// ---------------------------------------------------------------------------
// transition condition
      A     M    151.6; // Amount
      O     M    120.6;
      A     #S2I.SFM39.I01; // Released
      AN    M    102.2;
      =     M    102.1;

// subphase evaluation
      L     MW   110;
      JL    A300;
      JU    COMM; // subphase  0:
      JU    A301; // subphase  1: Gully VEE
      JU    A302; // subphase  2: Gully Befüllung
// ---------------------------------------------------------------------------
A300: SET   ;
      S     M    110.7; // Error unknown subphase
      JU    COMM;
// subphase 1: Gully VEE
A301: SET   ;
// -------------------------------------------------
// subphase timer & counter
      A     M    103.0;

// -------------------------------------------------
// subphase actuator
      A     M    103.3;

// -------------------------------------------------
// subphase transition
      SET   ;
      =     M    103.1;
      JU    COMM;
// subphase 2: Gully Befüllung
A302: SET   ;
// -------------------------------------------------
// subphase timer & counter
      A     M    103.0;

// -------------------------------------------------
// subphase actuator
      A     M    103.3;

// -------------------------------------------------
// subphase transition
      CLR   ;
      =     M    103.1;
      JU    COMM;

NETWORK
TITLE =phase 4: Fill System
//SFM   Use                                 Datatype        UoM
//----+-------------------------------------------------------------------------
// 00 : Watch Dog Time                      Duration        min
// 20 : Flow                                Value           l/h
// 41 : Amount                              Value           kg
X4:   SET   ;
// ---------------------------------------------------------------------------
// General CM evaluation
      CALL FC   120 (
           ChkType                  := 3,
           ChkOK                    := #ChkOK);

      AN    #ChkOK;
      S     M    120.3;

// ---------------------------------------------------------------------------
// general functions
      AN    M    121.2;
      A     M    102.3;
      =     #RRel;


// ---------------------------------------------------------------------------
// messages
// ---------------------------------------------------------------------------
// timer & counter
      A     M    102.0;

// ---------------------------------------------------------------------------
// pause timer
// ---------------------------------------------------------------------------
// communication

// ---------------------------------------------------------------------------
// control modules
      A     M    102.3;

// ---------------------------------------------------------------------------
// transition condition
      A     #SubStepMaxD;
      =     M    102.1;

// subphase evaluation
      L     MW   110;
      JL    A400;
      JU    COMM; // subphase  0:
// ---------------------------------------------------------------------------
A400: SET   ;
      S     M    110.7; // Error unknown subphase
      JU    COMM;

NETWORK
TITLE =phase 5: Transfer
//SFM   Use                                 Datatype        UoM
//----+-------------------------------------------------------------------------
// 00 : Watch Dog Time                      Duration        min
// 20 : Flow                                Value           l/h
// 41 : Amount                              Value           kg
X5:   SET   ;
// ---------------------------------------------------------------------------
// General CM evaluation
      CALL FC   120 (
           ChkType                  := 3,
           ChkOK                    := #ChkOK);

      AN    #ChkOK;
      S     M    120.3;

      CALL FC   779 (
           P1Sel                    := #U.Seq.SFM[11].Sp,
           P2Sel                    := #U.Seq.SFM[12].Sp,
           P3Sel                    := #U.Seq.SFM[13].Sp,
           P1Rel                    := DB125.DBX  363.2,
           P2Rel                    := DB125.DBX  411.2,
           P3Rel                    := DB125.DBX  459.2,
           CurrSel                  := #U.Seq.User.Real10);

// ---------------------------------------------------------------------------
// general functions
      AN    M    121.2;
      A     M    102.3;
      =     #RRel;

      A     M    102.3;
      =     DB125.DBX   26.3;

      A     M    102.3;
      =     DB125.DBX   27.2;

// ---------------------------------------------------------------------------
// messages

      AN    #ComDST;
      JCN   N501;
      L     903; // Destination not Ready
      T     MD    90;
N501: NOP   0;

// ---------------------------------------------------------------------------
// timer & counter

// Amount
      AN    #U.Seq.SFM[16].P;
      =     #xTmp;
      CALL FC   710 (
           RefVal                   := DB125.DBD  230,
           Active                   := #xTmp,
           Reset                    := #U.Seq.SFM[16].Res,
           Down                     := FALSE,
           CntVal                   := #U.Seq.SFM[16].Val,
           RefMem                   := #U.Seq.User.Real2);

      AN    #U.Seq.SFM[17].P; // TT Counter
      =     #xTmp;
      CALL FC   710 (
           RefVal                   := DB125.DBD  230,
           Active                   := #xTmp,
           Reset                    := #U.Seq.SFM[17].Res,
           Down                     := FALSE,
           CntVal                   := #U.Seq.SFM[17].Val,
           RefMem                   := #U.Seq.User.Real4);

// ---------------------------------------------------------------------------
// pause timer
// ---------------------------------------------------------------------------
// communication


// ---------------------------------------------------------------------------
// Check Partner
      AN    #ComSRC;
      O(    ;
      AN    DB125.DBX  218.3;
      AN    DB125.DBX  218.4;
      )     ;
      AN    #U.Seq.Step0;
      AN    #CIP;
      JCN   NC05;
      L     904; // "Source Not Ready!
      T     MD    90;
NC05: NOP   0;

      AN    DB125.DBX  314.0; // Water Tank Ready
      AN    DB125.DBX  314.1;
      AN    #ComDST;
      A     #S2I.SFM10.I00;
      AN    #U.Seq.Step0;
      AN    #U.Seq.PO.B22;
      AN    #CIP;
      JCN   NX05;
      L     903; // Destination not Ready
      T     MD    90;
NX05: NOP   0;

// ---------------------------------------------------------------------------
// control modules
      A     M    102.3;

// ---------------------------------------------------------------------------
// transition condition
      L     #U.Seq.User.Real10;
      L     0.000000e+000;
      ==R   ;
      O     M    151.7; // Amount
      AN    M    102.2;
      =     M    102.1;
// subphase repeat function
      A     #SubStepMax;
      JCN   Y5;
      L     1;
      T     MW   116;
Y5:   SET   ;
// ---------------------------------------------------------------------------
// ---------------------------------------------------------------------------
// subphase evaluation
      L     MW   110;
      JL    A500;
      JU    COMM; // subphase  0:
      JU    A501; // subphase  1: Waiting
      JU    A502; // subphase  2: Active
      JU    A503; // subphase  3: Tank Change
// ---------------------------------------------------------------------------
A500: SET   ;
      S     M    110.7; // Error unknown subphase
      JU    COMM;

// subphase 1: Waiting
A501: SET   ;

// -------------------------------------------------
// subphase timer & counter
      A     M    103.0;

// -------------------------------------------------
// subphase actuator
      A     M    103.3;

// -------------------------------------------------
// subphase transition
      A(    ;
      L     #U.Seq.User.Real10;
      L     #U.Seq.SFM[10].Sp;
      <>R   ;
      )     ;
      O(    ;
      A     DB125.DBX  314.0;
      A     DB125.DBX  315.2;
      A     DB125.DBX  218.3;
      O     #S2I.SFM10.I00;
      )     ;
      =     M    103.1;

      JU    COMM;

// subphase 2: Active
A502: SET   ;

// Well Management
      A     DB125.DBX  314.1;
      A     #ComSRC; // Comms Well Managment
      A     M    103.3;
      =     DB125.DBX   26.1; // Request Water

// Water Tank
      A     DB125.DBX  218.3; // Well Managment
      O     DB125.DBX  218.4; // Well Managment
      A     M    103.3;
      =     DB125.DBX   26.4;

// -------------------------------------------------
// subphase timer & counter
      A     M    103.0;
// -------------------------------------------------
// subphase actuator
      L     #U.Seq.SFM[22].Sp;
      L     1.000000e+001;
      <R    ;
      A(    ;
      L     #U.Seq.SFM[22].Sp;
      L     5.000000e+000;
      >R    ;
      )     ;
      A     DB125.DBX  314.1;
      A     DB125.DBX  219.7;
      A     M    103.3;
      =     DB220.DBX  348.0;
      =     DB220.DBX  188.0;
      =     DB220.DBX  268.0;
// -------------------------------------------------
// subphase transition
      L     #U.Seq.User.Real10;
      L     #U.Seq.SFM[10].Sp;
      <>R   ;
      O     #S2I.SFM10.I00;
      ON    DB125.DBX  315.2;
      =     M    103.1;

      JU    COMM;
// subphase 3: Tank Change
A503: SET   ;
      L     #U.Seq.User.Real10;
      T     #U.Seq.SFM[10].Sp; // Current Tank

// -------------------------------------------------
// subphase timer & counter
      A     M    103.0;
      =     M    162.0;

// -------------------------------------------------
// subphase actuator
//      A     "U099ComD".Own.Bit26
//      A     "SOSPH"
//      =     "C02ActD".A_G1.ACo
// -------------------------------------------------
// subphase transition
      AN    #S2I.SFM10.I00;
      AN    M    102.2;
      =     M    103.1;
      JU    COMM;
NETWORK
TITLE =phase 6: Standby
//SFM   Use                                 Datatype        UoM
//----+-------------------------------------------------------------------------
// 00 : Watch Dog Time                      Duration        min
// 02 : Step Time                           Duration        h
X6:   SET   ;
// ---------------------------------------------------------------------------
// General CM evaluation
      CALL FC   120 (
           ChkType                  := 3,
           ChkOK                    := #ChkOK);

      AN    #ChkOK;
      S     M    120.3;


      CALL FC   779 (
           P1Sel                    := #U.Seq.SFM[11].Sp,
           P2Sel                    := #U.Seq.SFM[12].Sp,
           P3Sel                    := #U.Seq.SFM[13].Sp,
           P1Rel                    := DB125.DBX  363.2,
           P2Rel                    := DB125.DBX  411.2,
           P3Rel                    := DB125.DBX  459.2,
           CurrSel                  := #U.Seq.User.Real10);

      L     #U.Seq.User.Real10;
      T     #U.Seq.SFM[10].Sp;

// ---------------------------------------------------------------------------
// general functions
      AN    M    121.2;
      A     M    102.3;
      =     #RRel;
      R     DB125.DBX   26.1;

      A     M    102.3;
      =     DB125.DBX   27.2;
// ---------------------------------------------------------------------------
// messages
      AN    M    151.7;
      A     M    150.1; // Max Standby Time
      JCN   N601;
      L     919; // "Press Start to Continue"
      T     MD    90;
N601: NOP   0;

// ---------------------------------------------------------------------------
// timer & counter
      A     M    102.0;
      =     M    130.1;
// ---------------------------------------------------------------------------
// pause timer
//      ON    "SOPH"
//      O     "SFM02D"
//      S     "SFM02P"                    // Step Time

      SET   ;
      S     M    141.7;

// ---------------------------------------------------------------------------
// communication

// ---------------------------------------------------------------------------
// Check Partner
      AN    #ComSRC;
      O(    ;
      AN    DB125.DBX  218.3;
      AN    DB125.DBX  218.4;
      )     ;
      AN    #U.Seq.Step0;
      AN    #CIP;
      JCN   NC06;
      L     904; // "Source Not Ready!
      T     MD    90;
NC06: NOP   0;

//      AN    "C02ComD".DST.WfFi          // Water Tank Ready
//      AN    "C02ComD".DST.Fill
      AN    #ComDST;
      AN    M    150.1; // Max Standby Time
//      A     #S2I.SFM10.I00
      AN    M    151.7;
      CLR   ; // Thats why we are in StandBy
      JCN   NX06;
      L     903; // Destination not Ready
      T     MD    90;
NX06: NOP   0;

// ---------------------------------------------------------------------------
// control modules

// ---------------------------------------------------------------------------
// transition condition
      CLR   ;
      =     #xTmp;

      AN    #S2I.SFM10.I00;
      AN    M    150.1; // Max Standby Time
      AN    M    151.7;
      S     #xTmp; // AutoCont
      JCN   N6x2;
      L     MW   104;
      L     -1;
      +I    ;
      T     MW   106;
N6x2: NOP   0;

      A     M    150.1; // Max Standby Time
      AN    M    151.7;
      A     M    120.6;
      S     #xTmp; // ReqRestart
      JCN   N6y2;
      L     MW   104;
      L     -2;
      +I    ;
      T     MW   106;
N6y2: NOP   0;

      A     M    150.1; // Max Standby Time
      A     M    151.7;
      S     #xTmp; // ReqEnd

      A     #xTmp;
      AN    M    102.2;
      =     M    102.1;

// subphase evaluation
      L     MW   110;
      JL    A600;
      JU    COMM; // subphase  0:
// ---------------------------------------------------------------------------
A600: SET   ;
      S     M    110.7; // Error unknown subphase
      JU    COMM;
NETWORK
TITLE =phase 8: Push Out
//SFM   Use                                 Datatype        UoM
//----+-------------------------------------------------------------------------
// 00 : Watch Dog Time                      Duration        min
// 20 : Flow                                Value           l/h
// 41 : Amount                              Value           kg
X8:   SET   ;
// ---------------------------------------------------------------------------
// General CM evaluation
      CALL FC   120 (
           ChkType                  := 3,
           ChkOK                    := #ChkOK);

      AN    #ChkOK;
      S     M    120.3;

// ---------------------------------------------------------------------------
// general functions
      AN    M    121.2;
      A     M    102.3;
      =     #RRel;

// ---------------------------------------------------------------------------
// messages
// ---------------------------------------------------------------------------
// timer & counter
      A     M    102.0;

// ---------------------------------------------------------------------------
// pause timer
// ---------------------------------------------------------------------------
// communication

// ---------------------------------------------------------------------------
// control modules
      A     M    102.3;

// ---------------------------------------------------------------------------
// transition condition
      A     #SubStepMaxD;
      =     M    102.1;

// subphase evaluation
      L     MW   110;
      JL    A800;
      JU    COMM; // subphase  0:
// ---------------------------------------------------------------------------
A800: SET   ;
      S     M    110.7; // Error unknown subphase
      JU    COMM;
NETWORK
TITLE =phase 11: Postrinse
//SFM   Use                                 Datatype        UoM
//----+-------------------------------------------------------------------------
// 00 : Watch Dog Time                      Duration        min
// 20 : Flow                                Value           l/h
// 41 : Amount                              Value           kg
X11:  SET   ;
// ---------------------------------------------------------------------------
// General CM evaluation
      CALL FC   120 (
           ChkType                  := 3,
           ChkOK                    := #ChkOK);

      AN    #ChkOK;
      S     M    120.3;

// ---------------------------------------------------------------------------
// general functions
      AN    M    121.2;
      A     M    102.3;
      =     #RRel;

// ---------------------------------------------------------------------------
// messages
// ---------------------------------------------------------------------------
// timer & counter
      A     M    102.0;

// ---------------------------------------------------------------------------
// pause timer
// ---------------------------------------------------------------------------
// communication

// ---------------------------------------------------------------------------
// control modules
      A     M    102.3;

// ---------------------------------------------------------------------------
// transition condition
      A     #SubStepMaxD;
      =     M    102.1;

// subphase evaluation
      L     MW   110;
      JL    B100;
      JU    COMM; // subphase  0:
// ---------------------------------------------------------------------------
B100: SET   ;
      S     M    110.7; // Error unknown subphase
      JU    COMM;
NETWORK
TITLE =phase 21: Prepare Line
//SFM   Use                                 Datatype        UoM
//----+-------------------------------------------------------------------------
// 00 : Watch Dog Time                      Duration        min
X21:  SET   ;
// ---------------------------------------------------------------------------
// General CM evaluation
      CALL FC   120 (
           ChkType                  := 3,
           ChkOK                    := #ChkOK);

      AN    #ChkOK;
      S     M    120.3;

      A     M    102.2;
      JCN   N903;
      L     DB125.DBD  234;
      T     #U.Seq.SFM[22].Sp;
N903: NOP   0;
// ---------------------------------------------------------------------------
// general functions
      AN    M    121.2;
      A     M    102.3;
      =     #RRel;

// ---------------------------------------------------------------------------
// messages
// ---------------------------------------------------------------------------
// timer & counter
      A     M    102.0;

// ---------------------------------------------------------------------------
// pause timer
// ---------------------------------------------------------------------------
// communication
      A     #ComSRC;
      A     M    103.3;
      =     DB125.DBX   26.0; // Wait for filling
      =     DB125.DBX   27.2;
// ---------------------------------------------------------------------------
// control modules
      A     M    102.3;

// ---------------------------------------------------------------------------
// transition condition
      A     #SubStepMaxD;
      AN    M    102.2;
      =     M    102.1;

// ---------------------------------------------------------------------------
// ---------------------------------------------------------------------------
// subphase repeat function
//      A     #SubStepMax
//      JCN  Y21
//      L     1
//      T     "SOSubStepNew"
//Y21:  SET

// subphase evaluation
      L     MW   110;
      JL    C100;
      JU    COMM; // subphase  0:
      JU    C101; // subphase  1: Start Well
      JU    C102; // subphase  2: Check Partner
// ---------------------------------------------------------------------------
C100: SET   ;
      S     M    110.7; // Error unknown subphase
      JU    COMM;

// subphase 1: Start Well
C101: SET   ;
// Request Well start

// -------------------------------------------------
// subphase timer & counter
      A     M    103.0;

// -------------------------------------------------
// subphase actuator
      A     M    103.3;

// -------------------------------------------------
// subphase transition
      A     DB125.DBX  218.3; // Well Ready
      A     #ComSRC;
      AN    M    103.2;
      =     M    103.1;
      JU    COMM;

// subphase 2: Check Partner
C102: SET   ;
      A     M    103.3;
      =     DB125.DBX   26.3;
// -------------------------------------------------
// subphase timer & counter
      A     M    103.0;

// -------------------------------------------------
// subphase actuator
      AN    DB125.DBX   75.2; // Swingbend drain Tank filling
      JCN   N801;
      L     920; // Check connections (Swingbend)
      T     MD    90;
N801: NOP   0;

// -------------------------------------------------
// subphase transition
      A     DB125.DBX   75.2; // Swingbend drain Tank filling
      A     DB125.DBX  218.3; // Well Ready
      A     #ComSRC; // Communication Well Management
      AN    M    103.2;
      =     M    103.1;
      JU    COMM;
NETWORK
TITLE =phase 22: Tank Selection
//SFM   Use                                 Datatype        UoM
//----+-------------------------------------------------------------------------
// 00 : Watch Dog Time                      Duration        min
X22:  SET   ;
// ---------------------------------------------------------------------------
// General CM evaluation
      CALL FC   120 (
           ChkType                  := 3,
           ChkOK                    := #ChkOK);

      AN    #ChkOK;
      S     M    120.3;

// ---------------------------------------------------------------------------
// general functions
      AN    M    121.2;
      A     M    102.3;
      =     #RRel;

// ---------------------------------------------------------------------------
// messages

      AN    #S2I.SFM11.I00; // Priority 1 Tank
      A     #ComSRC;
      JCN   N901;
      L     919; // "Press Start to Continue"
      T     MD    90;
N901: NOP   0;

// ---------------------------------------------------------------------------
// timer & counter
      A     M    102.0;

// ---------------------------------------------------------------------------
// pause timer
// ---------------------------------------------------------------------------
// communication
      A     M    102.0;
      R     DB125.DBX   26.1;
      A     M    102.0;
      =     DB125.DBX   26.0;

// ---------------------------------------------------------------------------
// control modules
      A     M    102.3;

// ---------------------------------------------------------------------------
// transition condition
      A     M    120.6;
      A     #ComSRC;
      AN    M    102.2;
      =     M    102.1;

// subphase evaluation
      L     MW   110;
      JL    C200;
      JU    COMM; // subphase  0:
// ---------------------------------------------------------------------------
C200: SET   ;
      S     M    110.7; // Error unknown subphase
      JU    COMM;

NETWORK
TITLE =End Of Sequence Organisation

COMM: SET   ;

// ---------------------------------------------------------------------------
// Comm with Transfer Plan Unit
      AN    DB125.DBX  509.0;
      R     DB125.DBX   29.0;

      L     DB125.DBD  510;
      L     #U.Seq.SFM[42].Sp;
      ==R   ;
      AN    DB125.DBX  504.7;
      AN    DB125.DBX   24.7;
      =     #ComPLN;

      A     DB125.DBX  509.0;
      AN    DB125.DBX   29.0;
      A     #ComPLN;
      A     M    102.3;
      JCN   CpDt;
      SET   ;
      =     DB125.DBX   29.0;
// Menge
      L     DB125.DBD  514;
      L     #U.Seq.SFM[16].E;
      -R    ;
      L     #U.Seq.SFM[16].Sp;
      +R    ;
      T     #U.Seq.SFM[16].Sp;

// Tanks
      L     #U.Seq.SFM[11].Sp;
      L     0.000000e+000;
      ==R   ;
      JCN   T1st;
      L     DB125.DBD  518;
      T     #U.Seq.SFM[11].Sp;
T1st: NOP   0;
      L     #U.Seq.SFM[12].Sp;
      L     0.000000e+000;
      ==R   ;
      JCN   T2st;
      L     DB125.DBD  518;
      T     #U.Seq.SFM[12].Sp;
T2st: NOP   0;
      L     #U.Seq.SFM[13].Sp;
      L     0.000000e+000;
      ==R   ;
      JCN   T3st;
      L     DB125.DBD  518;
      T     #U.Seq.SFM[13].Sp;
T3st: NOP   0;


CpDt: NOP   0;


NETWORK
TITLE =General Post Phase Controls

      NOP   0;

// ---------------------------------------------------------------------------
// general postphase controls
      AN    M    120.7;
      S     M    131.7;

// Check Selection / Material -----------------------------------------------
      L     0;
      L     DB125.DBD  318; // 1. Tank
      <R    ;
      JCN   MCk1;
      L     #U.Seq.SFM[42].Sp;
      <>R   ;
      S     M    120.3;
      JCN   MCk0;
      L     910;
      T     MD    80;
MCk0: NOP   0;
      L     0;
      L     DB125.DBD  366; // 1. Tank
      <R    ;
      JCN   MCk1;
      L     #U.Seq.SFM[42].Sp;
      <>R   ;
      JCN   MCk1;
      L     910;
      T     MD    90;
MCk1: NOP   0;
      L     0;
      L     DB125.DBD  414; // 2. Tank
      <R    ;
      JCN   MCk2;
      L     #U.Seq.SFM[42].Sp;
      <>R   ;
      JCN   MCk2;
      L     910;
      T     MD    90;
MCk2: NOP   0;
      L     0;
      L     DB125.DBD  462; // 3. Tank
      <R    ;
      JCN   MCk3;
      L     #U.Seq.SFM[42].Sp;
      <>R   ;
      JCN   MCk3;
      L     910;
      T     MD    90;
MCk3: NOP   0;

      L     #U.Seq.SFM[11].Sp;
      L     #U.Seq.SFM[12].Sp;
      OD    ;
      L     #U.Seq.SFM[13].Sp;
      OD    ;
      L     0;
      >R    ;
      O     M    120.7;
      JC    TSel;
      A     #S2I.SFM11.I00;
      L     905; // "Destination not Selected"
      T     MD    90;
TSel: NOP   0;

NETWORK
TITLE =Process Status Management

      NOP   0;
// ---------------------------------------------------------------------------
// Signal Control

      OPN   DB   500;
      L     #UnitNo;
      L     32; //U Structure Length
      *I    ;
      L     20; //DB Heading Offset
      +I    ;
      SLD   3;
      LAR2  ;

// -------------------------------------------------
// Maintenance
      A     #U.Seq.Switch.Sw31;
      OPN   DB   500;
      =     DBX [AR2,P#0.0]; //"PStatD".U[#UnitNo].MTNC
// -------------------------------------------------
// CIP Required
// -------------------------------------------------
// CIP Active
// -------------------------------------------------
// CIP Clean
// -------------------------------------------------
// SIP Required
// -------------------------------------------------
// SIP Active
// -------------------------------------------------
// SIP Clean
// -------------------------------------------------
// Full
      A     DB125.DBX   26.2;
      OPN   DB   500;
      =     DBX [AR2,P#0.7]; //"PStatD".U[#UnitNo].FULL
// -------------------------------------------------
// Filling
      A     DB125.DBX   26.1;
      OPN   DB   500;
      =     DBX [AR2,P#1.0]; //"PStatD".U[#UnitNo].FILL
// -------------------------------------------------
// Ready For Filling
      A     DB125.DBX   26.0;
      OPN   DB   500;
      =     DBX [AR2,P#1.1]; //"PStatD".U[#UnitNo].RFFI
// -------------------------------------------------
// Empty
      A     DB125.DBX   26.5;
      OPN   DB   500;
      =     DBX [AR2,P#1.2]; //"PStatD".U[#UnitNo].EMTY
// -------------------------------------------------
// Emptying
      A     DB125.DBX   26.4;
      OPN   DB   500;
      =     DBX [AR2,P#1.3]; //"PStatD".U[#UnitNo].EMTI
// -------------------------------------------------
// Ready For Emptying
      A     DB125.DBX   26.3;
      OPN   DB   500;
      =     DBX [AR2,P#1.4]; //"PStatD".U[#UnitNo].RFEM
// -------------------------------------------------
// Reserved
//      A     #ComXYZ
//      OPN   "PStatD"
//      =     DBX [AR2,P#1.5]             //"PStatD".U[#UnitNo].RESV
// -------------------------------------------------
// Production
// -------------------------------------------------
// Used

// -------------------------------------------------
// PStat Function Call

      CALL FC   500 (
           UnitNo                   := #UnitNo,
           PStatModVal              := DB225.DBD  234);

NETWORK
TITLE =Unit Hold Request and Messages

      SET   ;

// ---------------------------------------------------------------------------
// Set unit to "hold" if maintenance
      AN    #U.Seq.Switch.Sw31; // maintenance !
      JC    NCO1;
      S     M    120.3;
      L     998; // "Unit in maintenance !"
      T     MD    90;

// ---------------------------------------------------------------------------
// Set unit to "hold" if emergency stop
NCO1: A     #EStopOK;
      JC    NCO2;
      S     M    120.3;
      L     999; // "Emergency stop !"
      T     MD    90;
NCO2: NOP   0;





END_FUNCTION_BLOCK

FUNCTION_BLOCK FB 123
TITLE =C02: Well Transfer x
AUTHOR : Woermann
FAMILY : BOTEC_F1
NAME : C02E
VERSION : 1.2
CODE_VERSION1


VAR
  U : UDT 121;
END_VAR
VAR_TEMP
  CIP : BOOL ;	//CIP active
  UNIM : BOOL ;	//Unit Not In Maintenance
  GenRel : BOOL ;	//general OK (emergency and maintenance OK)
  EStopOK : BOOL ;	//emergency OK
  UnitNo : INT ;	//unit number
  xTmp : BOOL ;	//Temporary Bool
  iTmp : INT ;	//Temporary INT
  rTmp : REAL ;	//Temporary REAL
  dTmp : DINT ;	//Temporary DINT (free for general use)
  RetValInt : INT ;	//return value
  ComCIP1 : BOOL ;	//CIP1 in use
  ComCIP3 : BOOL ;	//CIP3 in use
END_VAR
BEGIN
NETWORK
TITLE =General

      SET   ;
// Simulation ---------------------------------------------------------------
      A     #U.Seq.User.Bit63;
      CC    FB   129; // "C02Sim"
      A     #U.Seq.Sim;
      =     #U.Seq.User.Bit63; //Help bit for simulation

// get unit number ----------------------------------------------------------
      L     MB   112;
      T     #UnitNo;

// CIP ----------------------------------------------------------------------
      L     #U.Seq.ProgNo;
      L     0;
      <D    ;
      =     #CIP;

// emergency OK -------------------------------------------------------------
      A     DB125.DBX   27.0; //Emergency Stop OK
      =     #EStopOK;

// Write Unit in Maintenance ------------------------------------------------

      AN    #U.Seq.Switch.Sw31;
      =     #UNIM;

// emergency and maintenance OK ---------------------------------------------
      A     #EStopOK;
      A     #UNIM;
      =     #GenRel;

// communication ------------------------------------------------------------
      UC    FB   125; // C02Com

NETWORK
TITLE =Analog Inputs

      NOP   0;

// ----------------------------------------------------------
// U31_AnI001 J6F_Druck
// ----------------------------------------------------------
      L     #U.Seq.SFM[63].Sp; // !!! insert correct SFM !!!
      T     DB223.DBD  238;

      SET   ;
      =     DB223.DBX  141.5;

// ----------------------------------------------------------
// QI_CO2_J6F_PH
// ----------------------------------------------------------
      L     #U.Seq.SFM[15].Sp;
      T     DB223.DBD  358;

      SET   ;
      =     DB223.DBX  261.5;

// ----------------------------------------------------------
// U31_AnI003 spare
// ----------------------------------------------------------
      L     #U.Seq.SFM[63].Sp; // !!! insert correct SFM !!!
      T     DB223.DBD  478;

      SET   ;
      =     DB223.DBX  381.5;

NETWORK
TITLE =Universal Value

      NOP   0;

// ----------------------------------------------------------
// unv001 Process Status
// ----------------------------------------------------------
// process value to UnV
//      L     0.000000e+000
//      T     "C02UnVD".unv001.ValExt

// ----------------------------------------------------------
// unv002 Universal Value 02
// ----------------------------------------------------------
// process value to UnV
      L     0.000000e+000;
      T     DB225.DBD  362;

// ----------------------------------------------------------
// unv003 Universal Value 03
// ----------------------------------------------------------
// process value to UnV
      SET   ;
      =     DB225.DBX  403.5;

// ----------------------------------------------------------
// unv004 Universal Value 04
// ----------------------------------------------------------
// process value to UnV
//      L     0.000000e+000
//      T     "C02UnVD".unv004.ValExt

NETWORK
TITLE =Special Input

      NOP   0;

// ----------------------------------------------------------
// U31_SpI001 spare
// ----------------------------------------------------------
      CLR   ; // Only used in one well?
      =     DB221.DBX   81.4;
      =     DB221.DBX   81.5;

// ----------------------------------------------------------
// U31_SpI002 spare
// ----------------------------------------------------------
      CLR   ; // Only used in one well?
      =     DB221.DBX  141.4;
      =     DB221.DBX  141.5;

// ----------------------------------------------------------
// U31_SpI003 spare
// ----------------------------------------------------------
      CLR   ; // Only used in one well?
      =     DB221.DBX  201.4;
      =     DB221.DBX  201.5;

NETWORK
TITLE =Messages

      NOP   0;

// ----------------------------------------------------------
// msg001 Message 01
// ----------------------------------------------------------
      SET   ;
      R     DB227.DBX   80.7;
      =     DB227.DBX   81.4;

      CLR   ;
      =     DB227.DBX   82.7;

// ----------------------------------------------------------
// msg002 Message 02
// ----------------------------------------------------------
      SET   ;
      R     DB227.DBX  140.7;
      =     DB227.DBX  141.4;

      CLR   ;
      =     DB227.DBX  142.7;

// ----------------------------------------------------------
// msg003 Message 03
// ----------------------------------------------------------
      SET   ;
      R     DB227.DBX  200.7;
      =     DB227.DBX  201.4;

      CLR   ;
      =     DB227.DBX  202.7;

NETWORK
TITLE =PID controller
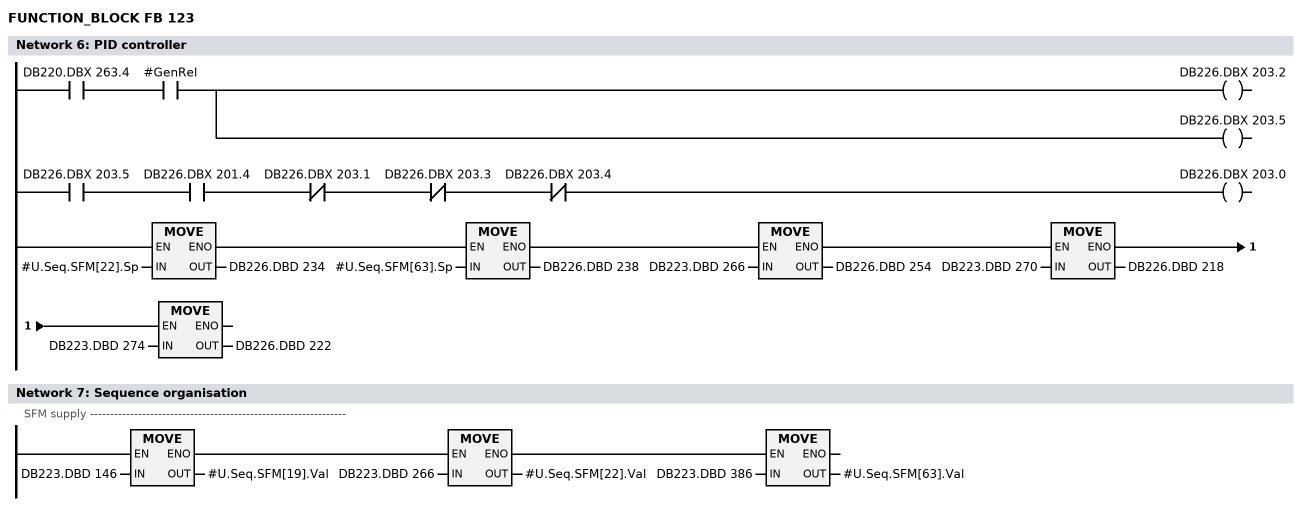

      NOP   0;

// ----------------------------------------------------------
// CO2J6FRV1 CO2 J6F RV1
// ----------------------------------------------------------
// starting value -----------------------
      A     DB220.DBX  263.4;
      A     #GenRel;
      =     DB226.DBX  203.2;
      =     DB226.DBX  203.5;

// enable alarm -------------------------
      A     DB226.DBX  203.5;
      A     DB226.DBX  201.4;
      AN    DB226.DBX  203.1;
      AN    DB226.DBX  203.3;
      AN    DB226.DBX  203.4;
      =     DB226.DBX  203.0;

// setpoint to controller ---------------
      L     #U.Seq.SFM[22].Sp;
      T     DB226.DBD  234;

// static value to controller ----------
      L     #U.Seq.SFM[63].Sp;
      T     DB226.DBD  238;

// process value to controller ----------
      L     DB223.DBD  266;
      T     DB226.DBD  254;

// low/high value to controller ---------
      L     DB223.DBD  270;
      T     DB226.DBD  218;

      L     DB223.DBD  274;
      T     DB226.DBD  222;

NETWORK
TITLE =Sequence organisation
//
// SFM supply ----------------------------------------------------------------

// analog value to SFM J6F_Druck -----------------------
      L     DB223.DBD  146;
      T     #U.Seq.SFM[19].Val;

// analog value to SFM QI_CO2_J6F_PH -------------------
      L     DB223.DBD  266;
      T     #U.Seq.SFM[22].Val;

// analog value to SFM spare -----------------------
      L     DB223.DBD  386;
      T     #U.Seq.SFM[63].Val; // !!! insert correct SFM !!! PH after CO2


NETWORK
TITLE =Auto / Manual

      SET   ;
      AN    M    122.2;
      JC    MODE;
      AN    M    120.1;

// assign actuator mode
      AN    M    120.1;
      =     DB220.DBX  105.4;
      =     DB220.DBX  185.4;
      =     DB220.DBX  265.4;
      =     DB220.DBX  345.4;

// assign PID mode
      S     DB226.DBX  201.4;
      S     DB226.DBX  201.5;

MODE: SET   ;

NETWORK
TITLE =J6F_G1 J6F_G1
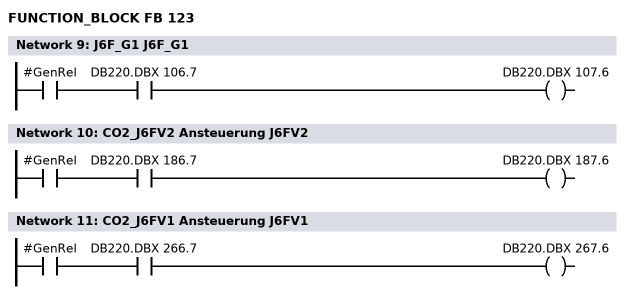

      A     #GenRel;
      A     DB220.DBX  106.7;
      =     DB220.DBX  107.6;
NETWORK
TITLE =CO2_J6FV2 Ansteuerung J6FV2

      A     #GenRel;
      A     DB220.DBX  186.7;
      =     DB220.DBX  187.6;
NETWORK
TITLE =CO2_J6FV1 Ansteuerung J6FV1

      A     #GenRel;
      A     DB220.DBX  266.7;
      =     DB220.DBX  267.6;
END_FUNCTION_BLOCK

FUNCTION_BLOCK FB 125
TITLE =C02: Well Transfer x
AUTHOR : Woermann
FAMILY : BOTEC_F1
NAME : C02Comm
VERSION : 0.1
CODE_VERSION1


VAR
  U : UDT 121;
END_VAR
VAR_TEMP
  iRetVal : INT ;	//return value as integer
  wRetVal : WORD ;	//return value as word
  Run : BOOL ;	//Unit in "RUN" mode
  EStopOK : BOOL ;	//Emergency Stop OK
  CIP : BOOL ;	//CIP Program Selected
  ComCIP : BOOL ;	//Communication with CIP Active
  xTmp : BOOL ;	//Temporary BOOL (free for general use)
  iTmp : INT ;	//Temporary INT (free for general use)
  rTmp : REAL ;	//Temporary REAL (free for general use)
  dTmp : DINT ;	//Temporary DINT (free for general use)
  UnitNo : INT ;	//Unit Number
  EquipmentID : INT ;	//Equipment ID
  Prid : DINT ;	//Process ID
  SFM36 : STRUCT 	//CIP Pump Mode
   I00 : BOOL ;	// Off
   I01 : BOOL ;	// Flow
   I02 : BOOL ;	// Pressure
   I03 : BOOL ;	// Fix Speed
   I04 : BOOL ;
   I05 : BOOL ;
   I06 : BOOL ;
   I07 : BOOL ;
   I08 : BOOL ;
   I09 : BOOL ;
   I10 : BOOL ;
   I11 : BOOL ;
   I12 : BOOL ;
   I13 : BOOL ;
   I14 : BOOL ;
   I15 : BOOL ;
   I16 : BOOL ;
   I17 : BOOL ;
   I18 : BOOL ;
   I19 : BOOL ;
   I20 : BOOL ;
   I21 : BOOL ;
   I22 : BOOL ;
   I23 : BOOL ;
   I24 : BOOL ;
   I25 : BOOL ;
   I26 : BOOL ;
   I27 : BOOL ;
   I28 : BOOL ;
   I29 : BOOL ;
   I30 : BOOL ;
   I31 : BOOL ;
  END_STRUCT ;
  iPLC : INT ;
  iUnit : INT ;
  rUnitNo : REAL ;
  DSTUnit : INT ;	//Destination Unit
  SRCUnit : INT ;
  rUnitNo_1 : REAL ;	//Unit Number Real
END_VAR
BEGIN
NETWORK
TITLE =general

      SET   ;

// unit & equipment number ---------------------------------------------------
      L     #U.Seq.UnitNo;
      T     #UnitNo;

      L     DB125.DBW   14;
      L     1000;
      *I    ;
      L     #UnitNo;
      +I    ;
      T     #EquipmentID;

// CIP ----------------------------------------------------------------------
      L     DB125.DBW   18;
      L     0;
      <I    ;
      =     #CIP;

// Communicating Units-------------------------------------------------------
      L     DB125.DBD   10;
      L     DB125.DBD  106;
      ==D   ;
      =     #ComCIP;

// emergency OK -------------------------------------------------------------
      A     DB125.DBX   75.0; //General Emergency Stop OK
      =     #EStopOK;

NETWORK
TITLE =read other unit's data

      SET   ;

// ... General Unit ----------/
      CALL SFC   20 (
           SRCBLK                   := DB1995.Own,
           RET_VAL                  := #iTmp,
           DSTBLK                   := DB125.GEN);

      A     DB125.DBX   75.0; //General Emergency Stop OK
      =     #EStopOK;

// ... CIP Unit ------------- /

      CALL FC   563 (
           ActReq                   := M    101.0,
           PLCNo                    := 3,
           SourceUnitNo             := 91,
           IsTUnit                  := FALSE,
           DstComDRec               := DB125.CIP,
           RET_VAL                  := #wRetVal);

//----------------------------------------
// Communication Well Management
//----------------------------------------
      L     #U.Seq.Prop.Index0; // Source
      ITD   ;
      DTR   ;
      T     #rTmp;

      CALL FC   950 (
           EquipmentNo              := #rTmp,
           PLCNo                    := #iPLC,
           UnitNo                   := #iUnit);

      L     #iUnit;
      L     25;
      ==I   ;
      JCN   U025;
      CALL SFC   20 (
           SRCBLK                   := DB1995.P04U025,
           RET_VAL                  := #iTmp,
           DSTBLK                   := DB125.SRC);
U025: NOP   0;

      L     #iUnit;
      L     26;
      ==I   ;
      JCN   U026;
      CALL SFC   20 (
           SRCBLK                   := DB1995.P04U026,
           RET_VAL                  := #iTmp,
           DSTBLK                   := DB125.SRC);
U026: NOP   0;

      L     #iUnit;
      L     27;
      ==I   ;
      JCN   U027;
      CALL SFC   20 (
           SRCBLK                   := DB1995.P04U027,
           RET_VAL                  := #iTmp,
           DSTBLK                   := DB125.SRC);
U027: NOP   0;

      L     #iUnit;
      L     28;
      ==I   ;
      JCN   U028;
      CALL SFC   20 (
           SRCBLK                   := DB1995.P04U028,
           RET_VAL                  := #iTmp,
           DSTBLK                   := DB125.SRC);
U028: NOP   0;

      L     #iUnit;
      L     29;
      ==I   ;
      JCN   U029;
      CALL SFC   20 (
           SRCBLK                   := DB1995.P04U029,
           RET_VAL                  := #iTmp,
           DSTBLK                   := DB125.SRC);
U029: NOP   0;

      L     #iUnit;
      L     30;
      ==I   ;
      JCN   U030;
      CALL SFC   20 (
           SRCBLK                   := DB1995.P04U030,
           RET_VAL                  := #iTmp,
           DSTBLK                   := DB125.SRC);
U030: NOP   0;

      L     #iUnit;
      L     31;
      ==I   ;
      JCN   U031;
      CALL SFC   20 (
           SRCBLK                   := DB1995.P04U031,
           RET_VAL                  := #iTmp,
           DSTBLK                   := DB125.SRC);
U031: NOP   0;

      L     #iUnit;
      L     32;
      ==I   ;
      JCN   U032;
      CALL SFC   20 (
           SRCBLK                   := DB1995.P04U032,
           RET_VAL                  := #iTmp,
           DSTBLK                   := DB125.SRC);
U032: NOP   0;

      L     #iUnit;
      L     33;
      ==I   ;
      JCN   U033;
      CALL SFC   20 (
           SRCBLK                   := DB1995.P04U033,
           RET_VAL                  := #iTmp,
           DSTBLK                   := DB125.SRC);
U033: NOP   0;

      L     #iUnit;
      L     34;
      ==I   ;
      JCN   U034;
      CALL SFC   20 (
           SRCBLK                   := DB1995.P04U034,
           RET_VAL                  := #iTmp,
           DSTBLK                   := DB125.SRC);
U034: NOP   0;


//----------------------------------------
// Communication Water Tank
//----------------------------------------
// Current Tank ----------------------------
      CALL FC   950 (
           EquipmentNo              := #U.Seq.SFM[10].Sp,
           PLCNo                    := #iPLC,
           UnitNo                   := #iUnit);

      L     #U.Seq.SFM[10].Sp;
      L     0.000000e+000;
      >R    ;
      JCN   N201;

      CALL FC   563 (
           ActReq                   := M    101.0,
           PLCNo                    := #iPLC,
           SourceUnitNo             := #iUnit,
           IsTUnit                  := FALSE,
           DstComDRec               := DB125.DST,
           RET_VAL                  := #wRetVal);
      JU    N2x1;
N201: NOP   0;
      L     0;
      T     #rTmp;
      CALL SFC   21 (
           BVAL                     := #rTmp,
           RET_VAL                  := #iTmp,
           BLK                      := DB125.DST);
N2x1: NOP   0;
// Priority 1 -----------------------------
      CALL FC   950 (
           EquipmentNo              := #U.Seq.SFM[11].Sp,
           PLCNo                    := #iPLC,
           UnitNo                   := #iUnit);

      L     #U.Seq.SFM[11].Sp;
      L     0.000000e+000;
      >R    ;
      JCN   N202;

      CALL FC   563 (
           ActReq                   := M    101.0,
           PLCNo                    := #iPLC,
           SourceUnitNo             := #iUnit,
           IsTUnit                  := FALSE,
           DstComDRec               := DB125.DST1,
           RET_VAL                  := #wRetVal);
      JU    N2x2;
N202: NOP   0;
      L     0;
      T     #rTmp;
      CALL SFC   21 (
           BVAL                     := #rTmp,
           RET_VAL                  := #iTmp,
           BLK                      := DB125.DST1);
N2x2: NOP   0;

// Priority 2 ----------------------------
      CALL FC   950 (
           EquipmentNo              := #U.Seq.SFM[12].Sp,
           PLCNo                    := #iPLC,
           UnitNo                   := #iUnit);

      L     #U.Seq.SFM[12].Sp;
      L     0.000000e+000;
      >R    ;
      JCN   N203;

      CALL FC   563 (
           ActReq                   := M    101.0,
           PLCNo                    := #iPLC,
           SourceUnitNo             := #iUnit,
           IsTUnit                  := FALSE,
           DstComDRec               := DB125.DST2,
           RET_VAL                  := #wRetVal);
      JU    N2x3;
N203: NOP   0;
      L     0;
      T     #rTmp;
      CALL SFC   21 (
           BVAL                     := #rTmp,
           RET_VAL                  := #iTmp,
           BLK                      := DB125.DST2);
N2x3: NOP   0;

// Priority 3 ----------------------------
      CALL FC   950 (
           EquipmentNo              := #U.Seq.SFM[13].Sp,
           PLCNo                    := #iPLC,
           UnitNo                   := #iUnit);

      L     #U.Seq.SFM[13].Sp;
      L     0.000000e+000;
      >R    ;
      JCN   N204;

      CALL FC   563 (
           ActReq                   := M    101.0,
           PLCNo                    := #iPLC,
           SourceUnitNo             := #iUnit,
           IsTUnit                  := FALSE,
           DstComDRec               := DB125.DST3,
           RET_VAL                  := #wRetVal);
      JU    N2x4;
N204: NOP   0;
      L     0;
      T     #rTmp;
      CALL SFC   21 (
           BVAL                     := #rTmp,
           RET_VAL                  := #iTmp,
           BLK                      := DB125.DST3);
N2x4: NOP   0;

// Plan ----------------------------
      L     #UnitNo;
      L     100;
      +I    ;
      T     #iUnit;

      CALL FC   563 (
           ActReq                   := M    101.0,
           PLCNo                    := 3,
           SourceUnitNo             := #iUnit,
           IsTUnit                  := FALSE,
           DstComDRec               := DB125.PLN,
           RET_VAL                  := #wRetVal);


NETWORK
TITLE =external releases

      SET   ;
      =     DB220.DBX  106.7;
      =     DB220.DBX  186.7;
      =     DB220.DBX  266.7;
      =     DB220.DBX  346.7;
NETWORK
TITLE =write own unit data

      SET   ;
//-- CIP Communication ---------------------------------------
      AN    #U.Seq.Step0;
      AN    #U.Seq.PO.B30; // CIP Active (Slave)
      A     #ComCIP;
      JCN   NCIP;
//Conductivity CIP Return
      L     DB125.DBD  150;
      T     #U.Seq.SFM[32].Val;

//Temperature CIP Return
      L     DB125.DBD  146;
      T     #U.Seq.SFM[30].Val;

//CIP Prerun Pump SP

      CALL FC    45 (
           SFM                      := #U.Seq.SFM[36].Sp,
           Indexes                  := #SFM36);


      L     0.000000e+000;
      A     #SFM36.I01;
      =     DB125.DBX  171.7;
      JCN   pfc;
      L     #U.Seq.SFM[34].Sp;
pfc:  NOP   0;
      A     #SFM36.I02;
      =     DB125.DBX  172.0;
      JCN   ppc;
      L     #U.Seq.SFM[35].Sp;
ppc:  NOP   0;
      A     #SFM36.I03;
      =     DB125.DBX  171.6;
      JCN   pxc;
      L     #U.Seq.SFM[29].Sp;
pxc:  NOP   0;
      T     DB125.DBD  182;

//CIP Return
      L     #U.Seq.SFM[28].Sp;
      T     DB125.DBD  186;
      L     DB125.DBD  138;
      T     #U.Seq.SFM[28].Val;

//CIP Prerun
      L     #U.Seq.SFM[27].Sp;
      T     DB125.DBD  190;
      L     DB125.DBD  142;
      T     #U.Seq.SFM[27].Val;

// Write Own Data to CIP
      L     DB125.DBD   10;
      T     DB125.DBD  154;

      L     DB125.DBW   14;
      T     DB125.DBW  158;

      L     DB125.DBW   16;
      T     DB125.DBW  160;

      L     DB125.DBW   18;
      T     DB125.DBW  162;

      L     DB125.DBW   20;
      T     DB125.DBW  164;

      L     DB125.DBW   22;
      T     DB125.DBW  166;

      A     DB125.DBX   24.0;
      =     DB125.DBX  168.0;

      A     DB125.DBX   24.1;
      =     DB125.DBX  168.1;

      A     DB125.DBX   24.2;
      =     DB125.DBX  168.2;

      A     DB125.DBX   24.3;
      =     DB125.DBX  168.3;

      A     DB125.DBX   24.4;
      =     DB125.DBX  168.4;

      A     DB125.DBX   24.5;
      =     DB125.DBX  168.5;

      A     DB125.DBX   24.6;
      =     DB125.DBX  168.6;

      A     DB125.DBX   24.7;
      =     DB125.DBX  168.7;

// Copy Data to CIP
      CALL SFC   20 (
           SRCBLK                   := DB125.ToCIP,
           RET_VAL                  := #iRetVal,
           DSTBLK                   := DB125.ToCIP);

NCIP: NOP   0;

//Empty Signal
//A     "C02SpID".SpI.Sig //!!!! Insert correct Empty Signal !!!
      CLR   ;
      =     DB125.DBX   26.5;

//Full Signal
//A     "C02SpID".SpI.Sig //!!!! Insert correct Full Signal !!!
      CLR   ;
      =     DB125.DBX   26.2;

//CIP Program Selected
      A     #CIP;
      =     DB125.DBX   27.1;

// Emergency Stop
      A     #EStopOK; //If needed add or replace with own SpI
      =     DB125.DBX   27.0; //Emergency Stop OK

// Material
      L     #U.Seq.SFM[42].Sp; // Material
      T     DB125.DBD   30;

      L     DB125.DBD  230;
      T     #U.Seq.User.Real3;

//----------------------------------------
// Communication Water Tank
//----------------------------------------

      L     #U.Seq.SFM[10].Sp; // Current Tank
      T     DB125.DBD   34;

      L     #U.Seq.SFM[11].Sp; // Tank Priority 1
      T     DB125.DBD   38;

      L     #U.Seq.SFM[12].Sp; // Tank Priority 2
      T     DB125.DBD   42;

      L     #U.Seq.SFM[13].Sp; // Tank Priority 3
      T     DB125.DBD   46;

NETWORK
TITLE = read from other unit data


//------------------------------------------------------

      CALL FC    29 (
           UnitNo                   := #UnitNo,
           Value                    := DB125.DBD  222,
           Enable                   := #U.Seq.PO.B4,
           Down                     := FALSE,
           OriginDetect             := 5.000000e-001,
           MaxDiffPS                := 1.000000e+000,
           SFMRec                   := #U.Seq.SFM[41],
           ValueOld                 := #U.Seq.User.Real0);


END_FUNCTION_BLOCK

FUNCTION_BLOCK FB 129
TITLE =C02: Well Transfer x
AUTHOR : Woermann
FAMILY : BOTEC_F1
NAME : C02Sim
VERSION : 0.1
CODE_VERSION1


VAR
  U : UDT 121;
END_VAR
VAR_TEMP
  CIP : BOOL ;	//CIP active
  xTmp : BOOL ;	//Temporary BOOL (free for general use)
  iTmp : INT ;	//Temporary INT (free for general use)
  rTmp : REAL ;	//Temporary REAL (free for general use)
  UnitNo : INT ;	//Unit Number
END_VAR
BEGIN
NETWORK
TITLE =General

      SET   ;
// get unit number ----------------------------------------------------------
      L     #U.Seq.UnitNo;
      T     #UnitNo;

// CIP ----------------------------------------------------------------------
      L     MW   114;
      L     0;
      <D    ;
      =     #CIP;

NETWORK
TITLE =Actuator

      A     #U.Seq.Sim;
      =     DB220.DBX  105.3;
      =     DB220.DBX  185.3;
      =     DB220.DBX  265.3;
      =     DB220.DBX  345.3;


NETWORK
TITLE =Special Input

      A     #U.Seq.Sim;
      =     DB221.DBX   81.3;
      =     DB221.DBX  141.3;
      =     DB221.DBX  201.3;

NETWORK
TITLE =Counter

      A     #U.Seq.Sim;
      A     M    101.0;
      CLR   ;
NETWORK
TITLE =Analog Input

      A     #U.Seq.Sim;
      =     DB223.DBX  141.3;
      =     DB223.DBX  261.3;
      =     DB223.DBX  381.3;
NETWORK
TITLE =Universal Value

      A     #U.Seq.Sim;
      =     DB225.DBX  149.3;
      =     DB225.DBX  277.3;
      =     DB225.DBX  405.3;
      =     DB225.DBX  533.3;

NETWORK
TITLE =PID

      A     #U.Seq.Sim;
      CLR   ;
      =     DB226.DBX  201.3;

NETWORK
TITLE =Message

      A     #U.Seq.Sim;
//      =     "C02MsgD".msg001.Sim;
//      =     "C02MsgD".msg002.Sim;
//      =     "C02MsgD".msg003.Sim;

NETWORK
TITLE =VLT

      A     #U.Seq.Sim;

END_FUNCTION_BLOCK

FUNCTION_BLOCK FB 131
TITLE =C03: Local Well Transfer x
// NW  1 : phase and index evaluation
// NW  2 : phase  1: start position
// NW  3 : phase  3: Prerinse
// NW  4 : phase  4: Fill System
// NW  5 : phase  5: Transfer
// NW  6 : phase  8: Push Out
// NW  7 : phase 11: Postrinse
// NW  8 : phase 21: Prepare Line
// NW  9 : phase 22: Tank Selection
// NW 10 : end of sequence
// NW 11 : unit hold request
//SFM   Use                                 Datatype        UoM
//----+-------------------------------------------------------------------------
// 09 : Process Time                        Duration        min
// 40 : Density                             Value           kg/l
// 42 : Material                            Value
// 43 : Destination                         Enumeration
// 44 : Standby                             Value
AUTHOR : Woermann
NAME : C03Seq
VERSION : 0.1
CODE_VERSION1


VAR
  U : UDT 131;
END_VAR
VAR_TEMP
  CIP : BOOL ;	//CIP active
  ComCIP : BOOL ;	//Communication With CIP Active
  ComWell : BOOL ;	//Communication With Local Well x
  RRel : BOOL ;	//Run Release
  EStopOK : BOOL ;	//emergency OK
  StepMax : BOOL ;	//StepMax (last) active
  SubStepMax : BOOL ;	//SubStepMax (last) active
  SubStepMaxD : BOOL ;	//SubStepMax (last) done
  ChkOK : BOOL ;	//SubStepMax (last) done
  xTmp : BOOL ;	//Temporary BOOL (free for general use)
  iTmp : INT ;	//Temporary INT (free for general use)
  dTmp : DINT ;	//Temporary DINT (free for general use)
  rTmp : REAL ;	//Temporary REAL (free for general use)
  dUnitNo : DINT ;	//Unit Number
  UnitNo : INT ;	//Unit Number
  EquipmentID : INT ;	//Equipment ID
  S2I : STRUCT 	//SFM to indexes
   SFM26 : STRUCT 	//Cip Step On Condition
    I00 : BOOL ;	//Please Select
    I01 : BOOL ;	//Conductivity High
    I02 : BOOL ;	//Conductivity Low
    I03 : BOOL ;	//Time
    I04 : BOOL ;	//Amount
    I05 : BOOL ;	//Temperature High
    I06 : BOOL ;	//Temperature Low
    I07 : BOOL ;
    I08 : BOOL ;
    I09 : BOOL ;
    I10 : BOOL ;
    I11 : BOOL ;
    I12 : BOOL ;
    I13 : BOOL ;
    I14 : BOOL ;
    I15 : BOOL ;
    I16 : BOOL ;
    I17 : BOOL ;
    I18 : BOOL ;
    I19 : BOOL ;
    I20 : BOOL ;
    I21 : BOOL ;
    I22 : BOOL ;
    I23 : BOOL ;
    I24 : BOOL ;
    I25 : BOOL ;
    I26 : BOOL ;
    I27 : BOOL ;
    I28 : BOOL ;
    I29 : BOOL ;
    I30 : BOOL ;
    I31 : BOOL ;
   END_STRUCT ;
   SFM27 : STRUCT 	//Cip Prerun
    I00 : BOOL ;	//None
    I01 : BOOL ;	//Recovered Water
    I02 : BOOL ;	//Caustic
    I03 : BOOL ;
    I04 : BOOL ;	//Acid
    I05 : BOOL ;
    I06 : BOOL ;
    I07 : BOOL ;
    I08 : BOOL ;
    I09 : BOOL ;
    I10 : BOOL ;
    I11 : BOOL ;
    I12 : BOOL ;	//Fresh Water
    I13 : BOOL ;	//Warm Water
    I14 : BOOL ;
    I15 : BOOL ;
    I16 : BOOL ;
    I17 : BOOL ;
    I18 : BOOL ;
    I19 : BOOL ;
    I20 : BOOL ;
    I21 : BOOL ;
    I22 : BOOL ;
    I23 : BOOL ;
    I24 : BOOL ;
    I25 : BOOL ;
    I26 : BOOL ;
    I27 : BOOL ;
    I28 : BOOL ;
    I29 : BOOL ;
    I30 : BOOL ;
    I31 : BOOL ;
   END_STRUCT ;
   SFM28 : STRUCT 	//Cip Return
    I00 : BOOL ;	//None
    I01 : BOOL ;	//Recovered Water
    I02 : BOOL ;	//Caustic
    I03 : BOOL ;
    I04 : BOOL ;	//Acid
    I05 : BOOL ;
    I06 : BOOL ;
    I07 : BOOL ;
    I08 : BOOL ;
    I09 : BOOL ;
    I10 : BOOL ;
    I11 : BOOL ;
    I12 : BOOL ;	//Fresh Water
    I13 : BOOL ;	//Warm Water
    I14 : BOOL ;
    I15 : BOOL ;	//Drain
    I16 : BOOL ;
    I17 : BOOL ;
    I18 : BOOL ;
    I19 : BOOL ;
    I20 : BOOL ;
    I21 : BOOL ;
    I22 : BOOL ;
    I23 : BOOL ;
    I24 : BOOL ;
    I25 : BOOL ;
    I26 : BOOL ;
    I27 : BOOL ;
    I28 : BOOL ;
    I29 : BOOL ;
    I30 : BOOL ;
    I31 : BOOL ;
   END_STRUCT ;
   SFM37 : STRUCT 	//Cip Pump Mode
    I00 : BOOL ;	//Off
    I01 : BOOL ;	//Flow
    I02 : BOOL ;	//Pressure
    I03 : BOOL ;	//Fix Speed
    I04 : BOOL ;
    I05 : BOOL ;
    I06 : BOOL ;
    I07 : BOOL ;
    I08 : BOOL ;
    I09 : BOOL ;
    I10 : BOOL ;
    I11 : BOOL ;
    I12 : BOOL ;
    I13 : BOOL ;
    I14 : BOOL ;
    I15 : BOOL ;
    I16 : BOOL ;
    I17 : BOOL ;
    I18 : BOOL ;
    I19 : BOOL ;
    I20 : BOOL ;
    I21 : BOOL ;
    I22 : BOOL ;
    I23 : BOOL ;
    I24 : BOOL ;
    I25 : BOOL ;
    I26 : BOOL ;
    I27 : BOOL ;
    I28 : BOOL ;
    I29 : BOOL ;
    I30 : BOOL ;
    I31 : BOOL ;
   END_STRUCT ;
   SFM31 : STRUCT 	//Cip Distribution Circuit No
    I00 : BOOL ;	//Please Select
    I01 : BOOL ;	//Auto Select
    I02 : BOOL ;
    I03 : BOOL ;
    I04 : BOOL ;
    I05 : BOOL ;
    I06 : BOOL ;
    I07 : BOOL ;
    I08 : BOOL ;
    I09 : BOOL ;
    I10 : BOOL ;
    I11 : BOOL ;
    I12 : BOOL ;
    I13 : BOOL ;
    I14 : BOOL ;
    I15 : BOOL ;
    I16 : BOOL ;
    I17 : BOOL ;
    I18 : BOOL ;
    I19 : BOOL ;
    I20 : BOOL ;
    I21 : BOOL ;
    I22 : BOOL ;
    I23 : BOOL ;
    I24 : BOOL ;
    I25 : BOOL ;
    I26 : BOOL ;
    I27 : BOOL ;
    I28 : BOOL ;
    I29 : BOOL ;
    I30 : BOOL ;
    I31 : BOOL ;
   END_STRUCT ;
   SFM39 : STRUCT 	//Q-Status
    I00 : BOOL ;	//Please select
    I01 : BOOL ;	//released
    I02 : BOOL ;
    I03 : BOOL ;
    I04 : BOOL ;
    I05 : BOOL ;
    I06 : BOOL ;	//Ignore
    I07 : BOOL ;
    I08 : BOOL ;
    I09 : BOOL ;	//locked
    I10 : BOOL ;
    I11 : BOOL ;
    I12 : BOOL ;
    I13 : BOOL ;
    I14 : BOOL ;
    I15 : BOOL ;
    I16 : BOOL ;
    I17 : BOOL ;
    I18 : BOOL ;
    I19 : BOOL ;
    I20 : BOOL ;
    I21 : BOOL ;
    I22 : BOOL ;
    I23 : BOOL ;
    I24 : BOOL ;
    I25 : BOOL ;
    I26 : BOOL ;
    I27 : BOOL ;
    I28 : BOOL ;
    I29 : BOOL ;
    I30 : BOOL ;
    I31 : BOOL ;
   END_STRUCT ;
   SFM10 : STRUCT 	//Current Tank
    I00 : BOOL ;	//Please Select
    I01 : BOOL ;	//Water Tank 1
    I02 : BOOL ;	//Water Tank 2
    I03 : BOOL ;	//Water Tank 2
    I04 : BOOL ;	//Water Tank 3
    I05 : BOOL ;	//Water Tank 4
    I06 : BOOL ;	//Water Tank 5
    I07 : BOOL ;	//Water Tank 6
    I08 : BOOL ;	//Water Tank 7
    I09 : BOOL ;	//Water Tank 8
    I10 : BOOL ;	//WAter Tank 9
    I11 : BOOL ;	//Water Tank 10
    I12 : BOOL ;	//Water Tank 11
    I13 : BOOL ;	//Water Tank 12
    I14 : BOOL ;	//Water Tank 13
    I15 : BOOL ;
    I16 : BOOL ;
    I17 : BOOL ;
    I18 : BOOL ;
    I19 : BOOL ;
    I20 : BOOL ;
    I21 : BOOL ;
    I22 : BOOL ;
    I23 : BOOL ;
    I24 : BOOL ;
    I25 : BOOL ;
    I26 : BOOL ;
    I27 : BOOL ;
    I28 : BOOL ;
    I29 : BOOL ;
    I30 : BOOL ;
    I31 : BOOL ;
   END_STRUCT ;
   SFM11 : STRUCT 	//1. Tank
    I00 : BOOL ;	//Please Select
    I01 : BOOL ;	//Water Tank 1
    I02 : BOOL ;	//Water Tank 2
    I03 : BOOL ;	//Water Tank 2
    I04 : BOOL ;	//Water Tank 3
    I05 : BOOL ;	//Water Tank 4
    I06 : BOOL ;	//Water Tank 5
    I07 : BOOL ;	//Water Tank 6
    I08 : BOOL ;	//Water Tank 7
    I09 : BOOL ;	//Water Tank 8
    I10 : BOOL ;	//WAter Tank 9
    I11 : BOOL ;	//Water Tank 10
    I12 : BOOL ;	//Water Tank 11
    I13 : BOOL ;	//Water Tank 12
    I14 : BOOL ;	//Water Tank 13
    I15 : BOOL ;
    I16 : BOOL ;
    I17 : BOOL ;
    I18 : BOOL ;
    I19 : BOOL ;
    I20 : BOOL ;
    I21 : BOOL ;
    I22 : BOOL ;
    I23 : BOOL ;
    I24 : BOOL ;
    I25 : BOOL ;
    I26 : BOOL ;
    I27 : BOOL ;
    I28 : BOOL ;
    I29 : BOOL ;
    I30 : BOOL ;
    I31 : BOOL ;
   END_STRUCT ;
   SFM12 : STRUCT 	//2. Tank
    I00 : BOOL ;	//Please Select
    I01 : BOOL ;	//Water Tank 1
    I02 : BOOL ;	//Water Tank 2
    I03 : BOOL ;	//Water Tank 2
    I04 : BOOL ;	//Water Tank 3
    I05 : BOOL ;	//Water Tank 4
    I06 : BOOL ;	//Water Tank 5
    I07 : BOOL ;	//Water Tank 6
    I08 : BOOL ;	//Water Tank 7
    I09 : BOOL ;	//Water Tank 8
    I10 : BOOL ;	//WAter Tank 9
    I11 : BOOL ;	//Water Tank 10
    I12 : BOOL ;	//Water Tank 11
    I13 : BOOL ;	//Water Tank 12
    I14 : BOOL ;	//Water Tank 13
    I15 : BOOL ;
    I16 : BOOL ;
    I17 : BOOL ;
    I18 : BOOL ;
    I19 : BOOL ;
    I20 : BOOL ;
    I21 : BOOL ;
    I22 : BOOL ;
    I23 : BOOL ;
    I24 : BOOL ;
    I25 : BOOL ;
    I26 : BOOL ;
    I27 : BOOL ;
    I28 : BOOL ;
    I29 : BOOL ;
    I30 : BOOL ;
    I31 : BOOL ;
   END_STRUCT ;
   SFM13 : STRUCT 	//3. Tank
    I00 : BOOL ;	//Please Select
    I01 : BOOL ;	//Water Tank 1
    I02 : BOOL ;	//Water Tank 2
    I03 : BOOL ;	//Water Tank 2
    I04 : BOOL ;	//Water Tank 3
    I05 : BOOL ;	//Water Tank 4
    I06 : BOOL ;	//Water Tank 5
    I07 : BOOL ;	//Water Tank 6
    I08 : BOOL ;	//Water Tank 7
    I09 : BOOL ;	//Water Tank 8
    I10 : BOOL ;	//WAter Tank 9
    I11 : BOOL ;	//Water Tank 10
    I12 : BOOL ;	//Water Tank 11
    I13 : BOOL ;	//Water Tank 12
    I14 : BOOL ;	//Water Tank 13
    I15 : BOOL ;
    I16 : BOOL ;
    I17 : BOOL ;
    I18 : BOOL ;
    I19 : BOOL ;
    I20 : BOOL ;
    I21 : BOOL ;
    I22 : BOOL ;
    I23 : BOOL ;
    I24 : BOOL ;
    I25 : BOOL ;
    I26 : BOOL ;
    I27 : BOOL ;
    I28 : BOOL ;
    I29 : BOOL ;
    I30 : BOOL ;
    I31 : BOOL ;
   END_STRUCT ;
   SFM23 : STRUCT 	//Chriwa 1
    I00 : BOOL ;	//Erstfiltart
    I01 : BOOL ;	//Aus
    I02 : BOOL ;	//Bereitschaft
    I03 : BOOL ;	//Stop
    I04 : BOOL ;	//Störung
    I05 : BOOL ;
    I06 : BOOL ;
    I07 : BOOL ;
    I08 : BOOL ;	//Betrieb
    I09 : BOOL ;	//Entspannen
    I10 : BOOL ;	//Absenken
    I11 : BOOL ;	//Spülen Luft
    I12 : BOOL ;	//Spülen Wasser/Luft
    I13 : BOOL ;	//Filterbettentleerung
    I14 : BOOL ;	//Spülen Wasser
    I15 : BOOL ;	//Affüllen
    I16 : BOOL ;	//Nicht definiert
    I17 : BOOL ;
    I18 : BOOL ;
    I19 : BOOL ;
    I20 : BOOL ;
    I21 : BOOL ;
    I22 : BOOL ;
    I23 : BOOL ;
    I24 : BOOL ;
    I25 : BOOL ;
    I26 : BOOL ;
    I27 : BOOL ;
    I28 : BOOL ;
    I29 : BOOL ;
    I30 : BOOL ;
    I31 : BOOL ;
   END_STRUCT ;
   SFM24 : STRUCT 	//Chriwa 2
    I00 : BOOL ;	//Erstfiltart
    I01 : BOOL ;	//Aus
    I02 : BOOL ;	//Bereitschaft
    I03 : BOOL ;	//Stop
    I04 : BOOL ;	//Störung
    I05 : BOOL ;
    I06 : BOOL ;
    I07 : BOOL ;
    I08 : BOOL ;	//Betrieb
    I09 : BOOL ;	//Entspannen
    I10 : BOOL ;	//Absenken
    I11 : BOOL ;	//Spülen Luft
    I12 : BOOL ;	//Spülen Wasser/Luft
    I13 : BOOL ;	//Filterbettentleerung
    I14 : BOOL ;	//Spülen Wasser
    I15 : BOOL ;	//Affüllen
    I16 : BOOL ;	//Nicht definiert
    I17 : BOOL ;
    I18 : BOOL ;
    I19 : BOOL ;
    I20 : BOOL ;
    I21 : BOOL ;
    I22 : BOOL ;
    I23 : BOOL ;
    I24 : BOOL ;
    I25 : BOOL ;
    I26 : BOOL ;
    I27 : BOOL ;
    I28 : BOOL ;
    I29 : BOOL ;
    I30 : BOOL ;
    I31 : BOOL ;
   END_STRUCT ;
  END_STRUCT ;
  ComCIPDist : BOOL ;	//Communication with CIP Distribution
  ComVE : BOOL ;	//Comminication with unit Water Treatment
  ComWTank2 : BOOL ;	//Communication Water Tank Priority 2
  comWTank3 : BOOL ;	//Communication Water Tank Priority 3
  comWTank1 : BOOL ;	//Communication Water Tank Priority 1
  ComSRC : BOOL ;	//Communication With Well
  ComDST : BOOL ;	//Communication with Water Tank
  CurrSel : REAL ;	//Current Tank Selection SP
  ComPLN : BOOL ;	//Communication with Transfer Plan
END_VAR
BEGIN
NETWORK
TITLE = Phase and Index Evaluation

      CLR   ;
      =     #RRel;
      =     DB135.DBX   29.0;

// ---------------------------------------------------------------------------
// write max used SFM's (last SFM number + 1)
      L     46;
      T     #U.SFMQuant;

// ---------------------------------------------------------------------------
// unit & equipment number
      L     MB   112;
      T     #UnitNo;

      L     DB135.DBW   14;
      L     1000;
      *I    ;
      L     #UnitNo;
      +I    ;
      T     #EquipmentID;

// ---------------------------------------------------------------------------
// CIP active
      L     MW   114;
      L     0;
      <I    ;
      =     #CIP;

// ---------------------------------------------------------------------------
// communicating units
      L     MD   124;
      L     DB135.DBD  106;
      ==D   ;
      =     #ComCIP;

      L     #U.Seq.SFM[42].Sp;
      L     DB135.DBD  318;
      ==D   ;
      =     #ComSRC;

      L     DB135.DBD  270; // Destination Material
      L     #U.Seq.SFM[42].Sp;
      ==R   ;
      =     #ComDST;

      L     DB135.DBD  366; // Destination Material
      L     #U.Seq.SFM[42].Sp;
      ==R   ;
      =     #comWTank1;

      L     DB135.DBD  414; // Destination Material
      L     #U.Seq.SFM[42].Sp;
      ==R   ;
      =     #ComWTank2;

      L     DB135.DBD  462; // Destination Material
      L     #U.Seq.SFM[42].Sp;
      ==R   ;
      =     #comWTank3;

      L     DB135.DBD  202;
      L     MD   124;
      ==D   ;
      A     DB135.DBX  218.0;
      =     #ComVE; // Water Treatment


// Load Source to SFM
      L     DB135.DBD  338;
      T     #U.Seq.SFM[14].Sp;

// ---------------------------------------------------------------------------
// process timer start
      SET   ;
      =     M    131.0;

// ---------------------------------------------------------------------------
// emergency OK
      A     DB135.DBX   27.0;
      =     #EStopOK;

// define last (Sub)Step active
      L     #U.Seq.StepMax;
      L     MW   104;
      ==I   ;
      =     #StepMax;

      L     #U.Seq.SubStepMax;
      L     MW   118;
      ==I   ;
      =     #SubStepMax;

      A     #SubStepMax;
      A     #U.Seq.SPD;
      AN    M    103.2;
      =     #SubStepMaxD;

// ---------------------------------------------------------------------------
// index evaluation: Current Tank
      CALL FC    45 (
           SFM                      := #U.Seq.SFM[10].Sp,
           Indexes                  := #S2I.SFM10);

// index evaluation: 1. Tank
      CALL FC    45 (
           SFM                      := #U.Seq.SFM[11].Sp,
           Indexes                  := #S2I.SFM11);

// index evaluation: 2. Tank
      CALL FC    45 (
           SFM                      := #U.Seq.SFM[12].Sp,
           Indexes                  := #S2I.SFM12);

// index evaluation: 3. Tank
      CALL FC    45 (
           SFM                      := #U.Seq.SFM[13].Sp,
           Indexes                  := #S2I.SFM13);

// index evaluation: Q-Status
      CALL FC    45 (
           SFM                      := #U.Seq.SFM[39].Sp,
           Indexes                  := #S2I.SFM39);


// index evaluation: Chriwa 1 Status
      CALL FC    45 (
           SFM                      := #U.Seq.SFM[23].Val,
           Indexes                  := #S2I.SFM23);
// index evaluation: Chriwa 2 Status
      CALL FC    45 (
           SFM                      := #U.Seq.SFM[24].Val,
           Indexes                  := #S2I.SFM24);

// ---------------------------------------------------------------------------
// phase evaluation
      L     MW   108;
      JL    X0;
      JU    X0; // phase  0:
      JU    X1; // phase  1: start position
      JU    X0; // phase  2:
      JU    X3; // phase  3: Prerinse
      JU    X4; // phase  4: Fill System
      JU    X5; // phase  5: Transfer
      JU    X6; // phase  6: Standby
      JU    X0; // phase  7:
      JU    X8; // phase  8: Push Out
      JU    X0; // phase  9:
      JU    X0; // phase 10:
      JU    X11; // phase 11: Postrinse
      JU    X0; // phase 12:
      JU    X0; // phase 13:
      JU    X0; // phase 14:
      JU    X0; // phase 15:
      JU    X0; // phase 16:
      JU    X0; // phase 17:
      JU    X0; // phase 18:
      JU    X0; // phase 19:
      JU    X0; // phase 20:
      JU    X21; // phase 21: Prepare Line
      JU    X22; // phase 22: Tank Selection
X0:   SET   ;
      S     M    108.7; // Error unknown phase
      JU    COMM;
NETWORK
TITLE =phase 1: startposition

X1:   SET   ;
// ---------------------------------------------------------------------------
// general functions
// ---------------------------------------------------------------------------
// reset signals
      A     M    102.2;
      R     #U.Seq.Switch.Sw1;
      R     #U.Seq.Switch.Sw2;
      R     DB135.DBX   26.1;

      L     0.000000e+000;
      T     DB135.DBD   30;
      T     DB135.DBD   34;
      T     DB135.DBD   38;
      T     DB135.DBD   42;
      T     DB135.DBD   50;
      T     DB135.DBD   54;
      T     #U.Seq.SFM[42].Sp; // Material
      T     #U.Seq.SFM[10].Sp; // Current Tank
      T     #U.Seq.SFM[11].Sp; // Priority 1
      T     #U.Seq.SFM[12].Sp; // Priority 2
      T     #U.Seq.SFM[13].Sp; // Priority 3

      AN    M    102.0;
      =     M    161.0; // Reset Process Timer

      CALL FC   709 (// Reset "Simulation" And "Ignore"
           UnitNo                   := #UnitNo,// Of All Control Modules
           Enable                   := M    102.2);// At First Cycle of Startposition (Idle)

// ---------------------------------------------------------------------------
// start check --------------------------------------------------------------
      A     #CIP;
      JC    M010;

      CALL FC   130 (
           ChkType                  := 1,// production
           ChkOK                    := M    122.0);
      JU    COMM;

M010: CALL FC   130 (
           ChkType                  := 2,// CIP
           ChkOK                    := M    122.0);
      JU    COMM;
NETWORK
TITLE =phase 3: Prerinse
//SFM   Use                                 Datatype        UoM
//----+-------------------------------------------------------------------------
// 00 : Watch Dog Time                      Duration        min
// 20 : Flow                                Value           l/h
// 41 : Amount                              Value           kg
X3:   SET   ;
// ---------------------------------------------------------------------------
// General CM evaluation
      CALL FC   130 (
           ChkType                  := 3,
           ChkOK                    := #ChkOK);

      AN    #ChkOK;
      S     M    120.3;

// ---------------------------------------------------------------------------
// general functions
      AN    M    121.2;
      A     M    102.3;
      =     #RRel;

      CALL FC   779 (
           P1Sel                    := #U.Seq.SFM[11].Sp,
           P2Sel                    := #U.Seq.SFM[12].Sp,
           P3Sel                    := #U.Seq.SFM[13].Sp,
           P1Rel                    := DB135.DBX  363.2,
           P2Rel                    := DB135.DBX  411.2,
           P3Rel                    := DB135.DBX  459.2,
           CurrSel                  := #U.Seq.User.Real10);

      L     #U.Seq.User.Real10;
      T     #U.Seq.SFM[10].Sp;

// ---------------------------------------------------------------------------
// messages
      A     #S2I.SFM39.I01; // Released
      JCN   N301;
      L     919; // "Press Start to Continue"
      T     MD    90;
N301: NOP   0;

      A     M    151.6; // Rinse Amount
      A     #S2I.SFM39.I00; // Please Select
      JCN   N302;
      L     816; // LAB Release Required
      T     MD    90;
N302: NOP   0;


// ---------------------------------------------------------------------------
// timer & counter
      A     M    102.0;
      =     M    131.6;

// Presinse
      AN    #U.Seq.SFM[15].P;
      =     #xTmp;
      CALL FC   710 (
           RefVal                   := DB135.DBD  326,
           Active                   := #xTmp,
           Reset                    := #U.Seq.SFM[15].Res,
           Down                     := FALSE,
           CntVal                   := #U.Seq.SFM[15].Val,
           RefMem                   := #U.Seq.User.Real1);

// ---------------------------------------------------------------------------
// pause timer  .
      SET   ;
      S     M    141.7;
// ---------------------------------------------------------------------------
// communication
// Water Tank
      A     M    102.3;
      =     DB135.DBX   26.3;
// Well Management

// ---------------------------------------------------------------------------
// control modules

// ---------------------------------------------------------------------------
// transition condition
      A     #SubStepMaxD;
      AN    M    102.2;
      =     M    102.1;

// subphase evaluation
      L     MW   110;
      JL    A300;
      JU    COMM; // subphase  0:
      JU    A301; // subphase  1: Gully VEE
      JU    A302; // subphase  2: Gully Befüllung
// ---------------------------------------------------------------------------
A300: SET   ;
      S     M    110.7; // Error unknown subphase
      JU    COMM;
// subphase 1: Gully VEE
A301: SET   ;
// -------------------------------------------------
// subphase timer & counter
      A     M    103.0;
      =     M    131.6;

      AN    M    151.6; // Rinse Amount
      A     M    103.3;
      =     DB135.DBX   26.1; // Request Water

      CLR   ;
      =     DB135.DBX   27.6;

// -------------------------------------------------
// subphase actuator
      AN    M    151.6;
      A     M    103.3;
      =     DB230.DBX  268.0;
      =     DB230.DBX  188.0;

// -------------------------------------------------
// subphase transition
      A     M    151.6;
      =     M    103.1;
      JU    COMM;
// subphase 2: Gully Befüllung
A302: SET   ;
// -------------------------------------------------
// subphase timer & counter
      A     M    103.0;
      =     M    131.6;

// Well
      A     DB135.DBX  218.0;
      AN    M    151.6; // Rinse Amount
      A     #ComSRC; // Comms Well
      A     M    103.3;
      =     DB135.DBX   27.6;

      A     DB135.DBX  218.1;
      AN    M    151.6; // Rinse Amount
      A     #ComSRC; // Comms Well
      A     M    103.3;
      =     DB135.DBX   26.1; // Request Water

// -------------------------------------------------
// subphase actuator
// Drain
      AN    DB135.DBX  218.1;
      AN    M    151.6;
      A     M    103.3;
      =     DB230.DBX  268.0;
      =     DB230.DBX  188.0;

      A     DB135.DBX  218.1;
      A     DB135.DBX   75.2;
      AN    M    151.6;
      A     M    103.3;
      =     DB230.DBX  108.0;

// -------------------------------------------------
// subphase transition
      A     M    151.6; // Amount
      O     M    120.6;
      A     #S2I.SFM39.I01; // Released
      AN    M    102.2;
      =     M    103.1;
      JU    COMM;

NETWORK
TITLE =phase 4: Fill System
//SFM   Use                                 Datatype        UoM
//----+-------------------------------------------------------------------------
// 00 : Watch Dog Time                      Duration        min
// 20 : Flow                                Value           l/h
// 41 : Amount                              Value           kg
X4:   SET   ;
// ---------------------------------------------------------------------------
// General CM evaluation
      CALL FC   130 (
           ChkType                  := 3,
           ChkOK                    := #ChkOK);

      AN    #ChkOK;
      S     M    120.3;

// ---------------------------------------------------------------------------
// general functions
      AN    M    121.2;
      A     M    102.3;
      =     #RRel;


// ---------------------------------------------------------------------------
// messages
// ---------------------------------------------------------------------------
// timer & counter
      A     M    102.0;

// ---------------------------------------------------------------------------
// pause timer
// ---------------------------------------------------------------------------
// communication

// ---------------------------------------------------------------------------
// control modules
      A     M    102.3;

// ---------------------------------------------------------------------------
// transition condition
      A     #SubStepMaxD;
      =     M    102.1;

// subphase evaluation
      L     MW   110;
      JL    A400;
      JU    COMM; // subphase  0:
// ---------------------------------------------------------------------------
A400: SET   ;
      S     M    110.7; // Error unknown subphase
      JU    COMM;
NETWORK
TITLE =phase 5: Transfer
//SFM   Use                                 Datatype        UoM
//----+-------------------------------------------------------------------------
// 00 : Watch Dog Time                      Duration        min
// 20 : Flow                                Value           l/h
// 41 : Amount                              Value           kg
X5:   SET   ;
// ---------------------------------------------------------------------------
// General CM evaluation
      CALL FC   130 (
           ChkType                  := 3,
           ChkOK                    := #ChkOK);

      AN    #ChkOK;
      S     M    120.3;

      CALL FC   779 (
           P1Sel                    := #U.Seq.SFM[11].Sp,
           P2Sel                    := #U.Seq.SFM[12].Sp,
           P3Sel                    := #U.Seq.SFM[13].Sp,
           P1Rel                    := DB135.DBX  363.2,
           P2Rel                    := DB135.DBX  411.2,
           P3Rel                    := DB135.DBX  459.2,
           CurrSel                  := #U.Seq.User.Real10);

// ---------------------------------------------------------------------------
// general functions
      AN    M    121.2;
      A     M    102.3;
      =     #RRel;

      A     M    102.3;
      =     DB135.DBX   26.3;
// ---------------------------------------------------------------------------
// messages


// ---------------------------------------------------------------------------
// timer & counter

// Amount
      AN    #U.Seq.SFM[16].P;
      =     #xTmp;
      CALL FC   710 (
           RefVal                   := DB135.DBD  326,
           Active                   := #xTmp,
           Reset                    := #U.Seq.SFM[16].Res,
           Down                     := FALSE,
           CntVal                   := #U.Seq.SFM[16].Val,
           RefMem                   := #U.Seq.User.Real2);

      AN    #U.Seq.SFM[17].P; // TT Counter
      =     #xTmp;
      CALL FC   710 (
           RefVal                   := DB135.DBD  326,
           Active                   := #xTmp,
           Reset                    := #U.Seq.SFM[17].Res,
           Down                     := FALSE,
           CntVal                   := #U.Seq.SFM[17].Val,
           RefMem                   := #U.Seq.User.Real4);

// ---------------------------------------------------------------------------
// pause timer
// ---------------------------------------------------------------------------
// communication

// ---------------------------------------------------------------------------
// control modules
      A     M    102.3;

// ---------------------------------------------------------------------------
// transition condition
      L     #U.Seq.User.Real10;
      L     0.000000e+000;
      ==R   ;
      O     M    151.7; // Amount
      AN    M    102.2;
      =     M    102.1;
// subphase repeat function
      A     #SubStepMax;
      JCN   Y5;
      L     1;
      T     MW   116;
Y5:   SET   ;
// ---------------------------------------------------------------------------
// ---------------------------------------------------------------------------
// subphase evaluation
      L     MW   110;
      JL    A500;
      JU    COMM; // subphase  0:
      JU    A501; // subphase  1: Waiting
      JU    A502; // subphase  2: Active
      JU    A503; // subphase  3: Tank Change
// ---------------------------------------------------------------------------
A500: SET   ;
      S     M    110.7; // Error unknown subphase
      JU    COMM;

// subphase 1: Waiting
A501: SET   ;
      A     M    103.3;
      =     DB135.DBX   26.0;
// -------------------------------------------------
// subphase timer & counter
      A     M    103.0;

// -------------------------------------------------
// subphase actuator
      A     M    103.3;

// -------------------------------------------------
// subphase transition
      A(    ;
      L     #U.Seq.User.Real10;
      L     #U.Seq.SFM[10].Sp;
      <>R   ;
      )     ;
      O(    ;
// A     "C03ComD".SRC.Bit26
      A     DB135.DBX  266.0;
      A     DB135.DBX  267.2;
      A     DB135.DBX  314.3;
      O     #S2I.SFM10.I00;
      )     ;
      A     #ComVE; // Water Treatment
      =     M    103.1;

      JU    COMM;

// subphase 2: Active
A502: SET   ;

// Well
      A     DB135.DBX  218.0;
      A     #ComSRC; // Comms Well
      A     M    103.3;
      =     DB135.DBX   27.6;

      A     DB135.DBX  266.0;
      O     DB135.DBX  266.1;
      A     DB135.DBX  218.1;
      A     #ComSRC; // Comms Well
      A     M    103.3;
      =     DB135.DBX   26.1; // Request Water

// Water Tank
      A     DB135.DBX  314.3; // Well
      O     DB135.DBX  314.4; // Well
      A     DB135.DBX  218.1; // neu 20230420
      A     M    103.3;
      =     DB135.DBX   26.4;

// -------------------------------------------------
// subphase timer & counter
      A     M    103.0;
// -------------------------------------------------
// subphase actuator
//    A     "C03ComD".SRC.WfEm          // Well Managment
//      O     "C03ComD".SRC.Emti          // Well Managment
//      A     "SOSPH"
//      =     "C03ActD".C03_Act002.ACo

// Drain
      AN    DB135.DBX  218.1;
      AN    M    151.6;
      A     M    103.3;
      CLR   ;
      =     DB230.DBX  268.0;
      =     DB230.DBX  188.0;

// -------------------------------------------------
// subphase transition
      L     #U.Seq.User.Real10;
      L     #U.Seq.SFM[10].Sp;
      <>R   ;
      O     #S2I.SFM10.I00;
      ON    #ComSRC;
      ON    #ComVE; // Water Treatment
      =     M    103.1;

      JU    COMM;
// subphase 3: Tank Change
A503: SET   ;
      L     #U.Seq.User.Real10;
      T     #U.Seq.SFM[10].Sp; // Current Tank

// -------------------------------------------------
// subphase timer & counter
      A     M    103.0;
      =     M    162.0;

// -------------------------------------------------
// subphase actuator
//      A     "U099ComD".Own.Bit26
//      A     "SOSPH"
//      =     "C03ActD".C03_Act001.ACo
// -------------------------------------------------
// subphase transition
      AN    #S2I.SFM10.I00;
      AN    M    102.2;
      =     M    103.1;
      JU    COMM;

NETWORK
TITLE =phase 6: Standby
//SFM   Use                                 Datatype        UoM
//----+-------------------------------------------------------------------------
// 00 : Watch Dog Time                      Duration        min
// 02 : Step Time                           Duration        h
X6:   SET   ;
// ---------------------------------------------------------------------------
// General CM evaluation
      CALL FC   130 (
           ChkType                  := 3,
           ChkOK                    := #ChkOK);

      AN    #ChkOK;
      S     M    120.3;

      CALL FC   779 (
           P1Sel                    := #U.Seq.SFM[11].Sp,
           P2Sel                    := #U.Seq.SFM[12].Sp,
           P3Sel                    := #U.Seq.SFM[13].Sp,
           P1Rel                    := DB135.DBX  363.2,
           P2Rel                    := DB135.DBX  411.2,
           P3Rel                    := DB135.DBX  459.2,
           CurrSel                  := #U.Seq.User.Real10);

      L     #U.Seq.User.Real10;
      T     #U.Seq.SFM[10].Sp;

// ---------------------------------------------------------------------------
// general functions
      AN    M    121.2;
      A     M    102.3;
      =     #RRel;
      R     DB135.DBX   26.1;

      A     M    102.3;
      =     DB135.DBX   27.2;
// ---------------------------------------------------------------------------
// messages
      AN    M    151.7;
      A     M    150.1; // Max Standby Time
      JCN   N601;
      L     919; // "Press Start to Continue"
      T     MD    90;
N601: NOP   0;

// ---------------------------------------------------------------------------
// timer & counter
      A     M    102.0;
      =     M    130.1;
// ---------------------------------------------------------------------------
// pause timer
//      ON    "SOPH"
//      O     "SFM02D"
//      S     "SFM02P"                    // Step Time

      SET   ;
      S     M    141.7;

// ---------------------------------------------------------------------------
// communication
      A     M    102.0;
      =     DB135.DBX   27.7; // Bereit für Rückspülen

// Check Partner
      AN    #ComSRC;
      O(    ;
      AN    DB135.DBX  314.3;
      AN    DB135.DBX  314.4;
      )     ;
      AN    #U.Seq.Step0;
      AN    #CIP;
      JCN   NC06;
      L     904; // "Source Not Ready!
      T     MD    90;
NC06: NOP   0;

      A     #S2I.SFM23.I02;
      A     #S2I.SFM24.I02;
      JC    NM01;
      L     913; // Wasseraufbereitung nicht bereit
      T     MD    90;
NM01: NOP   0;

// Rückspülen Wasseraufbereitung
      A     #S2I.SFM23.I00;
      O     #S2I.SFM24.I00;
      A     DB135.DBX  218.0;
      A     #ComSRC; // Comms Well
      A     M    103.3;
      =     DB135.DBX   27.6;
      =     DB135.DBX   26.1; // Request Water
      =     DB230.DBX  108.0;

// ---------------------------------------------------------------------------
// control moduless

// ---------------------------------------------------------------------------
// transition condition
      CLR   ;
      =     #xTmp;

      AN    #S2I.SFM10.I00;
      AN    M    150.1; // Max Standby Time
      AN    M    151.7;
      S     #xTmp; // AutoCont
      JCN   N6x2;
      L     MW   104;
      L     -1;
      +I    ;
      T     MW   106;
N6x2: NOP   0;

      A     M    150.1; // Max Standby Time
      AN    M    151.7;
      A     M    120.6;
      S     #xTmp; // ReqRestart
      JCN   N6y2;
      L     MW   104;
      L     -2;
      +I    ;
      T     MW   106;
N6y2: NOP   0;

      A     M    150.1; // Max Standby Time
      A     M    151.7;
      S     #xTmp; // ReqEnd

      A     #xTmp;
      AN    M    102.2;
      A     #S2I.SFM23.I02;
      A     #S2I.SFM24.I02;
      =     M    102.1;

// subphase evaluation
      L     MW   110;
      JL    A600;
      JU    COMM; // subphase  0:
// ---------------------------------------------------------------------------
A600: SET   ;
      S     M    110.7; // Error unknown subphase
      JU    COMM;
NETWORK
TITLE =phase 8: Push Out
//SFM   Use                                 Datatype        UoM
//----+-------------------------------------------------------------------------
// 00 : Watch Dog Time                      Duration        min
// 20 : Flow                                Value           l/h
// 41 : Amount                              Value           kg
X8:   SET   ;
// ---------------------------------------------------------------------------
// General CM evaluation
      CALL FC   130 (
           ChkType                  := 3,
           ChkOK                    := #ChkOK);

      AN    #ChkOK;
      S     M    120.3;

// ---------------------------------------------------------------------------
// general functions
      AN    M    121.2;
      A     M    102.3;
      =     #RRel;

// ---------------------------------------------------------------------------
// messages
// ---------------------------------------------------------------------------
// timer & counter
      A     M    102.0;

// ---------------------------------------------------------------------------
// pause timer
// ---------------------------------------------------------------------------
// communication

// ---------------------------------------------------------------------------
// control modules
      A     M    102.3;

// ---------------------------------------------------------------------------
// transition condition
      A     #SubStepMaxD;
      =     M    102.1;

// subphase evaluation
      L     MW   110;
      JL    A800;
      JU    COMM; // subphase  0:
// ---------------------------------------------------------------------------
A800: SET   ;
      S     M    110.7; // Error unknown subphase
      JU    COMM;
NETWORK
TITLE =phase 11: Postrinse
//SFM   Use                                 Datatype        UoM
//----+-------------------------------------------------------------------------
// 00 : Watch Dog Time                      Duration        min
// 20 : Flow                                Value           l/h
// 41 : Amount                              Value           kg
X11:  SET   ;
// ---------------------------------------------------------------------------
// General CM evaluation
      CALL FC   130 (
           ChkType                  := 3,
           ChkOK                    := #ChkOK);

      AN    #ChkOK;
      S     M    120.3;

// ---------------------------------------------------------------------------
// general functions
      AN    M    121.2;
      A     M    102.3;
      =     #RRel;

// ---------------------------------------------------------------------------
// messages
// ---------------------------------------------------------------------------
// timer & counter
      A     M    102.0;

// ---------------------------------------------------------------------------
// pause timer
// ---------------------------------------------------------------------------
// communication

// ---------------------------------------------------------------------------
// control modules
      A     M    102.3;

// ---------------------------------------------------------------------------
// transition condition
      A     #SubStepMaxD;
      =     M    102.1;

// subphase evaluation
      L     MW   110;
      JL    B100;
      JU    COMM; // subphase  0:
// ---------------------------------------------------------------------------
B100: SET   ;
      S     M    110.7; // Error unknown subphase
      JU    COMM;
NETWORK
TITLE =phase 21: Prepare Line
//SFM   Use                                 Datatype        UoM
//----+-------------------------------------------------------------------------
// 00 : Watch Dog Time                      Duration        min
X21:  SET   ;
// ---------------------------------------------------------------------------
// General CM evaluation
      CALL FC   130 (
           ChkType                  := 3,
           ChkOK                    := #ChkOK);

      AN    #ChkOK;
      S     M    120.3;

      A     M    102.2;
      JCN   N903;
      L     DB135.DBD  330;
      T     #U.Seq.SFM[22].Sp;
N903: NOP   0;
// ---------------------------------------------------------------------------
// general functions
      AN    M    121.2;
      A     M    102.3;
      =     #RRel;

// ---------------------------------------------------------------------------
// messages
// ---------------------------------------------------------------------------
// timer & counter
      A     M    102.0;

// ---------------------------------------------------------------------------
// pause timer
// ---------------------------------------------------------------------------
// communication
      A     #ComSRC;
      A     M    103.3;
      =     DB135.DBX   26.0; // Wait for filling
      =     DB135.DBX   27.2;

// ---------------------------------------------------------------------------
// control modules
      A     M    102.3;

// ---------------------------------------------------------------------------
// transition condition
      A     #SubStepMaxD;
      AN    M    102.2;
      =     M    102.1;

// ---------------------------------------------------------------------------
// ---------------------------------------------------------------------------
// subphase repeat function
//      A     #SubStepMax
//      JCN  Y21
//      L     1
//      T     "SOSubStepNew"
//Y21:  SET

// subphase evaluation
      L     MW   110;
      JL    C100;
      JU    COMM; // subphase  0:
      JU    C101; // subphase  1: Start Well
      JU    C102; // subphase  2: Check Partner
// ---------------------------------------------------------------------------
C100: SET   ;
      S     M    110.7; // Error unknown subphase
      JU    COMM;

// subphase 1: Start Well
C101: SET   ;
// Request Well start

// -------------------------------------------------
// subphase timer & counter
      A     M    103.0;

// -------------------------------------------------
// subphase actuator
      A     M    103.3;

// -------------------------------------------------
// subphase transition
      A     DB135.DBX  314.3; // Well Ready
      A     #ComSRC;
      AN    M    103.2;
      =     M    103.1;
      JU    COMM;

// subphase 2: Check Partner
C102: SET   ;
      A     M    103.3;
      =     DB135.DBX   26.3;
// -------------------------------------------------
// subphase timer & counter
      A     M    103.0;

// -------------------------------------------------
// subphase actuator
      AN    DB135.DBX   75.2; // Swingbend drain Tank filling
      JCN   N801;
      L     920; // Check connections (Swingbend)
      T     MD    90;
N801: NOP   0;

// -------------------------------------------------
// subphase transition
      A     DB135.DBX   75.2; // Swingbend drain Tank filling
      A     DB135.DBX  314.3; // Well Ready
      A     #ComSRC; // Communication Well Management
      A     #ComVE; // Water Treatment
      AN    M    103.2;
      =     M    103.1;
      JU    COMM;

NETWORK
TITLE =phase 22: Tank Selection
//SFM   Use                                 Datatype        UoM
//----+-------------------------------------------------------------------------
// 00 : Watch Dog Time                      Duration        min
X22:  SET   ;
// ---------------------------------------------------------------------------
// General CM evaluation
      CALL FC   130 (
           ChkType                  := 3,
           ChkOK                    := #ChkOK);

      AN    #ChkOK;
      S     M    120.3;

// ---------------------------------------------------------------------------
// general functions
      AN    M    121.2;
      A     M    102.3;
      =     #RRel;

// Load Source to SFM
      A     DB231.DBX   78.7;
      JCN   BR2A;
      L     4.001000e+003; // Well 2A
      JU    BR07;
BR2A: A     DB231.DBX  138.7;
      JCN   BR2B;
      L     4.002000e+003; // Well 2B
      JU    BR07;
BR2B: A     DB231.DBX  198.7;
      JCN   BR03;
      L     4.003000e+003; // Well 3
      JU    BR07;
BR03: A     DB231.DBX  258.7;
      JCN   BR07;
      L     4.004000e+003; // Well 7
      JU    BR07;
BR07: NOP   0;
      T     #U.Seq.SFM[14].Sp; // Source



// ---------------------------------------------------------------------------
// messages

      AN    #S2I.SFM11.I00; // Priority 1 Tank
      A     #ComSRC;
      JCN   N901;
      L     919; // "Press Start to Continue"
      T     MD    90;
N901: NOP   0;

// ---------------------------------------------------------------------------
// timer & counter
      A     M    102.0;

// ---------------------------------------------------------------------------
// pause timer
// ---------------------------------------------------------------------------
// communication
      A     M    102.0;
      R     DB135.DBX   26.1;
// ---------------------------------------------------------------------------
// control modules
      A     M    102.3;

// ---------------------------------------------------------------------------
// transition condition
      A     M    120.6;
      A     #ComSRC;
      AN    M    102.2;
      =     M    102.1;

// subphase evaluation
      L     MW   110;
      JL    C200;
      JU    COMM; // subphase  0:
// ---------------------------------------------------------------------------
C200: SET   ;
      S     M    110.7; // Error unknown subphase
      JU    COMM;

NETWORK
TITLE =End Of Sequence Organisation

COMM: SET   ;

// ---------------------------------------------------------------------------
// pause timer unit parameter
// Comm with Transfer Plan Unit
      AN    DB135.DBX  509.0;
      R     DB135.DBX   29.0;

      L     DB135.DBD  510;
      L     #U.Seq.SFM[42].Sp;
      ==R   ;
      AN    DB135.DBX  504.7;
      AN    DB135.DBX   24.7;
      =     #ComPLN;

      A     DB135.DBX  509.0;
      AN    DB135.DBX   29.0;
      A     #ComPLN;
      A     M    102.3;
      JCN   CpDt;
      SET   ;
      =     DB135.DBX   29.0;
// Menge
      L     DB135.DBD  514;
      L     #U.Seq.SFM[16].E;
      -R    ;
      L     #U.Seq.SFM[16].Sp;
      +R    ;
      T     #U.Seq.SFM[16].Sp;

// Tanks
      L     #U.Seq.SFM[11].Sp;
      L     0.000000e+000;
      ==R   ;
      JCN   T1st;
      L     DB135.DBD  518;
      T     #U.Seq.SFM[11].Sp;
T1st: NOP   0;
      L     #U.Seq.SFM[12].Sp;
      L     0.000000e+000;
      ==R   ;
      JCN   T2st;
      L     DB135.DBD  518;
      T     #U.Seq.SFM[12].Sp;
T2st: NOP   0;
      L     #U.Seq.SFM[13].Sp;
      L     0.000000e+000;
      ==R   ;
      JCN   T3st;
      L     DB135.DBD  518;
      T     #U.Seq.SFM[13].Sp;
T3st: NOP   0;


CpDt: NOP   0;


NETWORK
TITLE =General Post Phase Controls

      NOP   0;

// ---------------------------------------------------------------------------
// general postphase controls
      AN    M    120.7;
      S     M    131.7;

// Check Selection / Material -----------------------------------------------
      L     0;
      L     DB135.DBD  270; // 1. Tank
      <R    ;
      JCN   MCk1;
      L     #U.Seq.SFM[42].Sp;
      <>R   ;
      S     M    120.3;
      JCN   MCk0;
      L     910;
      T     MD    80;
MCk0: NOP   0;
      L     0;
      L     DB135.DBD  366; // 1. Tank
      <R    ;
      JCN   MCk1;
      L     #U.Seq.SFM[42].Sp;
      <>R   ;
      JCN   MCk1;
      L     910;
      T     MD    90;
MCk1: NOP   0;
      L     0;
      L     DB135.DBD  414; // 2. Tank
      <R    ;
      JCN   MCk2;
      L     #U.Seq.SFM[42].Sp;
      <>R   ;
      JCN   MCk2;
      L     910;
      T     MD    90;
MCk2: NOP   0;
      L     0;
      L     DB135.DBD  462; // 3. Tank
      <R    ;
      JCN   MCk3;
      L     #U.Seq.SFM[42].Sp;
      <>R   ;
      JCN   MCk3;
      L     910;
      T     MD    90;
MCk3: NOP   0;

      L     #U.Seq.SFM[11].Sp;
      L     #U.Seq.SFM[12].Sp;
      OD    ;
      L     #U.Seq.SFM[13].Sp;
      OD    ;
      L     0;
      >R    ;
      O     M    120.7;
      JC    TSel;
      A     #S2I.SFM11.I00;
      L     905; // "Destination not Selected"
      T     MD    90;
TSel: NOP   0;

NETWORK
TITLE =Process Status Management

      NOP   0;
// ---------------------------------------------------------------------------
// Signal Control

      OPN   DB   500;
      L     #UnitNo;
      L     32; //U Structure Length
      *I    ;
      L     20; //DB Heading Offset
      +I    ;
      SLD   3;
      LAR2  ;

